    // Linear interpolation: y = vlo*(1-t) + vhi*t
    vlo := lut_table[lo];
    vhi := lut_table[hi];
    t := (x - lut_grid[lo]) / (lut_grid[hi] - lut_grid[lo] + 1.0E-10);
    "BsplineEval" := vlo * (1.0 - t) + vhi * t;
END_FUNCTION

FUNCTION_BLOCK "NeuroPLC_Inference"
{ S7_Optimized_Access := 'TRUE' }
VERSION : 0.1
VAR_INPUT
    features : Array[0..27] of Real;
END_VAR

VAR_OUTPUT
    fault_class : Int;
    confidence : Real;
END_VAR

VAR
    i, j, k : Int;
    sum_val, max_val, t_val : Real;
    v0 : Array[0..27] of Real;
    v1 : Array[0..27] of Real;
    v3 : Array[0..15, 0..27] of Real;
    v2 : Array[0..15] of Real;
    v4 : Array[0..15] of Real;
    v5 : Array[0..15] of Real;
    v7 : Array[0..3, 0..15] of Real;
    v6 : Array[0..3] of Real;
    v8 : Array[0..3] of Real;
    v9 : Array[0..3] of Real;
    lut_tmp : Array[0..14] of Real;
END_VAR

BEGIN
    // ---- Input ----
    FOR i := 0 TO 27 DO
        v0[i] := features[i];
    END_FOR;

    // ---- l0_silu: SILU ----
    v1[0] := v0[0] / (1.0 + EXP(-v0[0]));
    v1[1] := v0[1] / (1.0 + EXP(-v0[1]));
    v1[2] := v0[2] / (1.0 + EXP(-v0[2]));
    v1[3] := v0[3] / (1.0 + EXP(-v0[3]));
    v1[4] := v0[4] / (1.0 + EXP(-v0[4]));
    v1[5] := v0[5] / (1.0 + EXP(-v0[5]));
    v1[6] := v0[6] / (1.0 + EXP(-v0[6]));
    v1[7] := v0[7] / (1.0 + EXP(-v0[7]));
    v1[8] := v0[8] / (1.0 + EXP(-v0[8]));
    v1[9] := v0[9] / (1.0 + EXP(-v0[9]));
    v1[10] := v0[10] / (1.0 + EXP(-v0[10]));
    v1[11] := v0[11] / (1.0 + EXP(-v0[11]));
    v1[12] := v0[12] / (1.0 + EXP(-v0[12]));
    v1[13] := v0[13] / (1.0 + EXP(-v0[13]));
    v1[14] := v0[14] / (1.0 + EXP(-v0[14]));
    v1[15] := v0[15] / (1.0 + EXP(-v0[15]));
    v1[16] := v0[16] / (1.0 + EXP(-v0[16]));
    v1[17] := v0[17] / (1.0 + EXP(-v0[17]));
    v1[18] := v0[18] / (1.0 + EXP(-v0[18]));
    v1[19] := v0[19] / (1.0 + EXP(-v0[19]));
    v1[20] := v0[20] / (1.0 + EXP(-v0[20]));
    v1[21] := v0[21] / (1.0 + EXP(-v0[21]));
    v1[22] := v0[22] / (1.0 + EXP(-v0[22]));
    v1[23] := v0[23] / (1.0 + EXP(-v0[23]));
    v1[24] := v0[24] / (1.0 + EXP(-v0[24]));
    v1[25] := v0[25] / (1.0 + EXP(-v0[25]));
    v1[26] := v0[26] / (1.0 + EXP(-v0[26]));
    v1[27] := v0[27] / (1.0 + EXP(-v0[27]));

    // ---- l0_bspline: BsplineLUT(28×16, 15pts) ----
    // φ[0→0]: evaluate LUT (table offset 0)
    FOR k := 0 TO 14 DO
        lut_tmp[k] := "NeuroPLC_Weights".w1[0 + k];
    END_FOR;
    v3[0, 0] := "BsplineEval"(x := v0[0], lut_grid := "NeuroPLC_Weights".w0, lut_table := lut_tmp);
    // φ[1→0]: evaluate LUT (table offset 15)
    FOR k := 0 TO 14 DO
        lut_tmp[k] := "NeuroPLC_Weights".w1[15 + k];
    END_FOR;
    v3[0, 1] := "BsplineEval"(x := v0[1], lut_grid := "NeuroPLC_Weights".w0, lut_table := lut_tmp);
    // φ[2→0]: evaluate LUT (table offset 30)
    FOR k := 0 TO 14 DO
        lut_tmp[k] := "NeuroPLC_Weights".w1[30 + k];
    END_FOR;
    v3[0, 2] := "BsplineEval"(x := v0[2], lut_grid := "NeuroPLC_Weights".w0, lut_table := lut_tmp);
    // φ[3→0]: evaluate LUT (table offset 45)
    FOR k := 0 TO 14 DO
        lut_tmp[k] := "NeuroPLC_Weights".w1[45 + k];
    END_FOR;
    v3[0, 3] := "BsplineEval"(x := v0[3], lut_grid := "NeuroPLC_Weights".w0, lut_table := lut_tmp);
    // φ[4→0]: evaluate LUT (table offset 60)
    FOR k := 0 TO 14 DO
        lut_tmp[k] := "NeuroPLC_Weights".w1[60 + k];
    END_FOR;
    v3[0, 4] := "BsplineEval"(x := v0[4], lut_grid := "NeuroPLC_Weights".w0, lut_table := lut_tmp);
    // φ[5→0]: evaluate LUT (table offset 75)
    FOR k := 0 TO 14 DO
        lut_tmp[k] := "NeuroPLC_Weights".w1[75 + k];
    END_FOR;
    v3[0, 5] := "BsplineEval"(x := v0[5], lut_grid := "NeuroPLC_Weights".w0, lut_table := lut_tmp);
    // φ[6→0]: evaluate LUT (table offset 90)
    FOR k := 0 TO 14 DO
        lut_tmp[k] := "NeuroPLC_Weights".w1[90 + k];
    END_FOR;
    v3[0, 6] := "BsplineEval"(x := v0[6], lut_grid := "NeuroPLC_Weights".w0, lut_table := lut_tmp);
    // φ[7→0]: evaluate LUT (table offset 105)
    FOR k := 0 TO 14 DO
        lut_tmp[k] := "NeuroPLC_Weights".w1[105 + k];
    END_FOR;
    v3[0, 7] := "BsplineEval"(x := v0[7], lut_grid := "NeuroPLC_Weights".w0, lut_table := lut_tmp);
    // φ[8→0]: evaluate LUT (table offset 120)
    FOR k := 0 TO 14 DO
        lut_tmp[k] := "NeuroPLC_Weights".w1[120 + k];
    END_FOR;
    v3[0, 8] := "BsplineEval"(x := v0[8], lut_grid := "NeuroPLC_Weights".w0, lut_table := lut_tmp);
    // φ[9→0]: evaluate LUT (table offset 135)
    FOR k := 0 TO 14 DO
        lut_tmp[k] := "NeuroPLC_Weights".w1[135 + k];
    END_FOR;
    v3[0, 9] := "BsplineEval"(x := v0[9], lut_grid := "NeuroPLC_Weights".w0, lut_table := lut_tmp);
    // φ[10→0]: evaluate LUT (table offset 150)
    FOR k := 0 TO 14 DO
        lut_tmp[k] := "NeuroPLC_Weights".w1[150 + k];
    END_FOR;
    v3[0, 10] := "BsplineEval"(x := v0[10], lut_grid := "NeuroPLC_Weights".w0, lut_table := lut_tmp);
    // φ[11→0]: evaluate LUT (table offset 165)
    FOR k := 0 TO 14 DO
        lut_tmp[k] := "NeuroPLC_Weights".w1[165 + k];
    END_FOR;
    v3[0, 11] := "BsplineEval"(x := v0[11], lut_grid := "NeuroPLC_Weights".w0, lut_table := lut_tmp);
    // φ[12→0]: evaluate LUT (table offset 180)
    FOR k := 0 TO 14 DO
        lut_tmp[k] := "NeuroPLC_Weights".w1[180 + k];
    END_FOR;
    v3[0, 12] := "BsplineEval"(x := v0[12], lut_grid := "NeuroPLC_Weights".w0, lut_table := lut_tmp);
    // φ[13→0]: evaluate LUT (table offset 195)
    FOR k := 0 TO 14 DO
        lut_tmp[k] := "NeuroPLC_Weights".w1[195 + k];
    END_FOR;
    v3[0, 13] := "BsplineEval"(x := v0[13], lut_grid := "NeuroPLC_Weights".w0, lut_table := lut_tmp);
    // φ[14→0]: evaluate LUT (table offset 210)
    FOR k := 0 TO 14 DO
        lut_tmp[k] := "NeuroPLC_Weights".w1[210 + k];
    END_FOR;
    v3[0, 14] := "BsplineEval"(x := v0[14], lut_grid := "NeuroPLC_Weights".w0, lut_table := lut_tmp);
    // φ[15→0]: evaluate LUT (table offset 225)
    FOR k := 0 TO 14 DO
        lut_tmp[k] := "NeuroPLC_Weights".w1[225 + k];
    END_FOR;
    v3[0, 15] := "BsplineEval"(x := v0[15], lut_grid := "NeuroPLC_Weights".w0, lut_table := lut_tmp);
    // φ[16→0]: evaluate LUT (table offset 240)
    FOR k := 0 TO 14 DO
        lut_tmp[k] := "NeuroPLC_Weights".w1[240 + k];
    END_FOR;
    v3[0, 16] := "BsplineEval"(x := v0[16], lut_grid := "NeuroPLC_Weights".w0, lut_table := lut_tmp);
    // φ[17→0]: evaluate LUT (table offset 255)
    FOR k := 0 TO 14 DO
        lut_tmp[k] := "NeuroPLC_Weights".w1[255 + k];
    END_FOR;
    v3[0, 17] := "BsplineEval"(x := v0[17], lut_grid := "NeuroPLC_Weights".w0, lut_table := lut_tmp);
    // φ[18→0]: evaluate LUT (table offset 270)
    FOR k := 0 TO 14 DO
        lut_tmp[k] := "NeuroPLC_Weights".w1[270 + k];
    END_FOR;
    v3[0, 18] := "BsplineEval"(x := v0[18], lut_grid := "NeuroPLC_Weights".w0, lut_table := lut_tmp);
    // φ[19→0]: evaluate LUT (table offset 285)
    FOR k := 0 TO 14 DO
        lut_tmp[k] := "NeuroPLC_Weights".w1[285 + k];
    END_FOR;
    v3[0, 19] := "BsplineEval"(x := v0[19], lut_grid := "NeuroPLC_Weights".w0, lut_table := lut_tmp);
    // φ[20→0]: evaluate LUT (table offset 300)
    FOR k := 0 TO 14 DO
        lut_tmp[k] := "NeuroPLC_Weights".w1[300 + k];
    END_FOR;
    v3[0, 20] := "BsplineEval"(x := v0[20], lut_grid := "NeuroPLC_Weights".w0, lut_table := lut_tmp);
    // φ[21→0]: evaluate LUT (table offset 315)
    FOR k := 0 TO 14 DO
        lut_tmp[k] := "NeuroPLC_Weights".w1[315 + k];
    END_FOR;
    v3[0, 21] := "BsplineEval"(x := v0[21], lut_grid := "NeuroPLC_Weights".w0, lut_table := lut_tmp);
    // φ[22→0]: evaluate LUT (table offset 330)
    FOR k := 0 TO 14 DO
        lut_tmp[k] := "NeuroPLC_Weights".w1[330 + k];
    END_FOR;
    v3[0, 22] := "BsplineEval"(x := v0[22], lut_grid := "NeuroPLC_Weights".w0, lut_table := lut_tmp);
    // φ[23→0]: evaluate LUT (table offset 345)
    FOR k := 0 TO 14 DO
        lut_tmp[k] := "NeuroPLC_Weights".w1[345 + k];
    END_FOR;
    v3[0, 23] := "BsplineEval"(x := v0[23], lut_grid := "NeuroPLC_Weights".w0, lut_table := lut_tmp);
    // φ[24→0]: evaluate LUT (table offset 360)
    FOR k := 0 TO 14 DO
        lut_tmp[k] := "NeuroPLC_Weights".w1[360 + k];
    END_FOR;
    v3[0, 24] := "BsplineEval"(x := v0[24], lut_grid := "NeuroPLC_Weights".w0, lut_table := lut_tmp);
    // φ[25→0]: evaluate LUT (table offset 375)
    FOR k := 0 TO 14 DO
        lut_tmp[k] := "NeuroPLC_Weights".w1[375 + k];
    END_FOR;
    v3[0, 25] := "BsplineEval"(x := v0[25], lut_grid := "NeuroPLC_Weights".w0, lut_table := lut_tmp);
    // φ[26→0]: evaluate LUT (table offset 390)
    FOR k := 0 TO 14 DO
        lut_tmp[k] := "NeuroPLC_Weights".w1[390 + k];
    END_FOR;
    v3[0, 26] := "BsplineEval"(x := v0[26], lut_grid := "NeuroPLC_Weights".w0, lut_table := lut_tmp);
    // φ[27→0]: evaluate LUT (table offset 405)
    FOR k := 0 TO 14 DO
        lut_tmp[k] := "NeuroPLC_Weights".w1[405 + k];
    END_FOR;
    v3[0, 27] := "BsplineEval"(x := v0[27], lut_grid := "NeuroPLC_Weights".w0, lut_table := lut_tmp);
    // φ[0→1]: evaluate LUT (table offset 420)
    FOR k := 0 TO 14 DO
        lut_tmp[k] := "NeuroPLC_Weights".w1[420 + k];
    END_FOR;
    v3[1, 0] := "BsplineEval"(x := v0[0], lut_grid := "NeuroPLC_Weights".w0, lut_table := lut_tmp);
    // φ[1→1]: evaluate LUT (table offset 435)
    FOR k := 0 TO 14 DO
        lut_tmp[k] := "NeuroPLC_Weights".w1[435 + k];
    END_FOR;
    v3[1, 1] := "BsplineEval"(x := v0[1], lut_grid := "NeuroPLC_Weights".w0, lut_table := lut_tmp);
    // φ[2→1]: evaluate LUT (table offset 450)
    FOR k := 0 TO 14 DO
        lut_tmp[k] := "NeuroPLC_Weights".w1[450 + k];
    END_FOR;
    v3[1, 2] := "BsplineEval"(x := v0[2], lut_grid := "NeuroPLC_Weights".w0, lut_table := lut_tmp);
    // φ[3→1]: evaluate LUT (table offset 465)
    FOR k := 0 TO 14 DO
        lut_tmp[k] := "NeuroPLC_Weights".w1[465 + k];
    END_FOR;
    v3[1, 3] := "BsplineEval"(x := v0[3], lut_grid := "NeuroPLC_Weights".w0, lut_table := lut_tmp);
    // φ[4→1]: evaluate LUT (table offset 480)
    FOR k := 0 TO 14 DO
        lut_tmp[k] := "NeuroPLC_Weights".w1[480 + k];
    END_FOR;
    v3[1, 4] := "BsplineEval"(x := v0[4], lut_grid := "NeuroPLC_Weights".w0, lut_table := lut_tmp);
    // φ[5→1]: evaluate LUT (table offset 495)
    FOR k := 0 TO 14 DO
        lut_tmp[k] := "NeuroPLC_Weights".w1[495 + k];
    END_FOR;
    v3[1, 5] := "BsplineEval"(x := v0[5], lut_grid := "NeuroPLC_Weights".w0, lut_table := lut_tmp);
    // φ[6→1]: evaluate LUT (table offset 510)
    FOR k := 0 TO 14 DO
        lut_tmp[k] := "NeuroPLC_Weights".w1[510 + k];
    END_FOR;
    v3[1, 6] := "BsplineEval"(x := v0[6], lut_grid := "NeuroPLC_Weights".w0, lut_table := lut_tmp);
    // φ[7→1]: evaluate LUT (table offset 525)
    FOR k := 0 TO 14 DO
        lut_tmp[k] := "NeuroPLC_Weights".w1[525 + k];
    END_FOR;
    v3[1, 7] := "BsplineEval"(x := v0[7], lut_grid := "NeuroPLC_Weights".w0, lut_table := lut_tmp);
    // φ[8→1]: evaluate LUT (table offset 540)
    FOR k := 0 TO 14 DO
        lut_tmp[k] := "NeuroPLC_Weights".w1[540 + k];
    END_FOR;
    v3[1, 8] := "BsplineEval"(x := v0[8], lut_grid := "NeuroPLC_Weights".w0, lut_table := lut_tmp);
    // φ[9→1]: evaluate LUT (table offset 555)
    FOR k := 0 TO 14 DO
        lut_tmp[k] := "NeuroPLC_Weights".w1[555 + k];
    END_FOR;
    v3[1, 9] := "BsplineEval"(x := v0[9], lut_grid := "NeuroPLC_Weights".w0, lut_table := lut_tmp);
    // φ[10→1]: evaluate LUT (table offset 570)
    FOR k := 0 TO 14 DO
        lut_tmp[k] := "NeuroPLC_Weights".w1[570 + k];
    END_FOR;
    v3[1, 10] := "BsplineEval"(x := v0[10], lut_grid := "NeuroPLC_Weights".w0, lut_table := lut_tmp);
    // φ[11→1]: evaluate LUT (table offset 585)
    FOR k := 0 TO 14 DO
        lut_tmp[k] := "NeuroPLC_Weights".w1[585 + k];
    END_FOR;
    v3[1, 11] := "BsplineEval"(x := v0[11], lut_grid := "NeuroPLC_Weights".w0, lut_table := lut_tmp);
    // φ[12→1]: evaluate LUT (table offset 600)
    FOR k := 0 TO 14 DO
        lut_tmp[k] := "NeuroPLC_Weights".w1[600 + k];
    END_FOR;
    v3[1, 12] := "BsplineEval"(x := v0[12], lut_grid := "NeuroPLC_Weights".w0, lut_table := lut_tmp);
    // φ[13→1]: evaluate LUT (table offset 615)
    FOR k := 0 TO 14 DO
        lut_tmp[k] := "NeuroPLC_Weights".w1[615 + k];
    END_FOR;
    v3[1, 13] := "BsplineEval"(x := v0[13], lut_grid := "NeuroPLC_Weights".w0, lut_table := lut_tmp);
    // φ[14→1]: evaluate LUT (table offset 630)
    FOR k := 0 TO 14 DO
        lut_tmp[k] := "NeuroPLC_Weights".w1[630 + k];
    END_FOR;
    v3[1, 14] := "BsplineEval"(x := v0[14], lut_grid := "NeuroPLC_Weights".w0, lut_table := lut_tmp);
    // φ[15→1]: evaluate LUT (table offset 645)
    FOR k := 0 TO 14 DO
        lut_tmp[k] := "NeuroPLC_Weights".w1[645 + k];
    END_FOR;
    v3[1, 15] := "BsplineEval"(x := v0[15], lut_grid := "NeuroPLC_Weights".w0, lut_table := lut_tmp);
    // φ[16→1]: evaluate LUT (table offset 660)
    FOR k := 0 TO 14 DO
        lut_tmp[k] := "NeuroPLC_Weights".w1[660 + k];
    END_FOR;
    v3[1, 16] := "BsplineEval"(x := v0[16], lut_grid := "NeuroPLC_Weights".w0, lut_table := lut_tmp);
    // φ[17→1]: evaluate LUT (table offset 675)
    FOR k := 0 TO 14 DO
        lut_tmp[k] := "NeuroPLC_Weights".w1[675 + k];
    END_FOR;
    v3[1, 17] := "BsplineEval"(x := v0[17], lut_grid := "NeuroPLC_Weights".w0, lut_table := lut_tmp);
    // φ[18→1]: evaluate LUT (table offset 690)
    FOR k := 0 TO 14 DO
        lut_tmp[k] := "NeuroPLC_Weights".w1[690 + k];
    END_FOR;
    v3[1, 18] := "BsplineEval"(x := v0[18], lut_grid := "NeuroPLC_Weights".w0, lut_table := lut_tmp);
    // φ[19→1]: evaluate LUT (table offset 705)
    FOR k := 0 TO 14 DO
        lut_tmp[k] := "NeuroPLC_Weights".w1[705 + k];
    END_FOR;
    v3[1, 19] := "BsplineEval"(x := v0[19], lut_grid := "NeuroPLC_Weights".w0, lut_table := lut_tmp);
    // φ[20→1]: evaluate LUT (table offset 720)
    FOR k := 0 TO 14 DO
        lut_tmp[k] := "NeuroPLC_Weights".w1[720 + k];
    END_FOR;
    v3[1, 20] := "BsplineEval"(x := v0[20], lut_grid := "NeuroPLC_Weights".w0, lut_table := lut_tmp);
    // φ[21→1]: evaluate LUT (table offset 735)
    FOR k := 0 TO 14 DO
        lut_tmp[k] := "NeuroPLC_Weights".w1[735 + k];
    END_FOR;
    v3[1, 21] := "BsplineEval"(x := v0[21], lut_grid := "NeuroPLC_Weights".w0, lut_table := lut_tmp);
    // φ[22→1]: evaluate LUT (table offset 750)
    FOR k := 0 TO 14 DO
        lut_tmp[k] := "NeuroPLC_Weights".w1[750 + k];
    END_FOR;
    v3[1, 22] := "BsplineEval"(x := v0[22], lut_grid := "NeuroPLC_Weights".w0, lut_table := lut_tmp);
    // φ[23→1]: evaluate LUT (table offset 765)
    FOR k := 0 TO 14 DO
        lut_tmp[k] := "NeuroPLC_Weights".w1[765 + k];
    END_FOR;
    v3[1, 23] := "BsplineEval"(x := v0[23], lut_grid := "NeuroPLC_Weights".w0, lut_table := lut_tmp);
    // φ[24→1]: evaluate LUT (table offset 780)
    FOR k := 0 TO 14 DO
        lut_tmp[k] := "NeuroPLC_Weights".w1[780 + k];
    END_FOR;
    v3[1, 24] := "BsplineEval"(x := v0[24], lut_grid := "NeuroPLC_Weights".w0, lut_table := lut_tmp);
    // φ[25→1]: evaluate LUT (table offset 795)
    FOR k := 0 TO 14 DO
        lut_tmp[k] := "NeuroPLC_Weights".w1[795 + k];
    END_FOR;
    v3[1, 25] := "BsplineEval"(x := v0[25], lut_grid := "NeuroPLC_Weights".w0, lut_table := lut_tmp);
    // φ[26→1]: evaluate LUT (table offset 810)
    FOR k := 0 TO 14 DO
        lut_tmp[k] := "NeuroPLC_Weights".w1[810 + k];
    END_FOR;
    v3[1, 26] := "BsplineEval"(x := v0[26], lut_grid := "NeuroPLC_Weights".w0, lut_table := lut_tmp);
    // φ[27→1]: evaluate LUT (table offset 825)
    FOR k := 0 TO 14 DO
        lut_tmp[k] := "NeuroPLC_Weights".w1[825 + k];
    END_FOR;
    v3[1, 27] := "BsplineEval"(x := v0[27], lut_grid := "NeuroPLC_Weights".w0, lut_table := lut_tmp);
    // φ[0→2]: evaluate LUT (table offset 840)
    FOR k := 0 TO 14 DO
        lut_tmp[k] := "NeuroPLC_Weights".w1[840 + k];
    END_FOR;
    v3[2, 0] := "BsplineEval"(x := v0[0], lut_grid := "NeuroPLC_Weights".w0, lut_table := lut_tmp);
    // φ[1→2]: evaluate LUT (table offset 855)
    FOR k := 0 TO 14 DO
        lut_tmp[k] := "NeuroPLC_Weights".w1[855 + k];
    END_FOR;
    v3[2, 1] := "BsplineEval"(x := v0[1], lut_grid := "NeuroPLC_Weights".w0, lut_table := lut_tmp);
    // φ[2→2]: evaluate LUT (table offset 870)
    FOR k := 0 TO 14 DO
        lut_tmp[k] := "NeuroPLC_Weights".w1[870 + k];
    END_FOR;
    v3[2, 2] := "BsplineEval"(x := v0[2], lut_grid := "NeuroPLC_Weights".w0, lut_table := lut_tmp);
    // φ[3→2]: evaluate LUT (table offset 885)
    FOR k := 0 TO 14 DO
        lut_tmp[k] := "NeuroPLC_Weights".w1[885 + k];
    END_FOR;
    v3[2, 3] := "BsplineEval"(x := v0[3], lut_grid := "NeuroPLC_Weights".w0, lut_table := lut_tmp);
    // φ[4→2]: evaluate LUT (table offset 900)
    FOR k := 0 TO 14 DO
        lut_tmp[k] := "NeuroPLC_Weights".w1[900 + k];
    END_FOR;
    v3[2, 4] := "BsplineEval"(x := v0[4], lut_grid := "NeuroPLC_Weights".w0, lut_table := lut_tmp);
    // φ[5→2]: evaluate LUT (table offset 915)
    FOR k := 0 TO 14 DO
        lut_tmp[k] := "NeuroPLC_Weights".w1[915 + k];
    END_FOR;
    v3[2, 5] := "BsplineEval"(x := v0[5], lut_grid := "NeuroPLC_Weights".w0, lut_table := lut_tmp);
    // φ[6→2]: evaluate LUT (table offset 930)
    FOR k := 0 TO 14 DO
        lut_tmp[k] := "NeuroPLC_Weights".w1[930 + k];
    END_FOR;
    v3[2, 6] := "BsplineEval"(x := v0[6], lut_grid := "NeuroPLC_Weights".w0, lut_table := lut_tmp);
    // φ[7→2]: evaluate LUT (table offset 945)
    FOR k := 0 TO 14 DO
        lut_tmp[k] := "NeuroPLC_Weights".w1[945 + k];
    END_FOR;
    v3[2, 7] := "BsplineEval"(x := v0[7], lut_grid := "NeuroPLC_Weights".w0, lut_table := lut_tmp);
    // φ[8→2]: evaluate LUT (table offset 960)
    FOR k := 0 TO 14 DO
        lut_tmp[k] := "NeuroPLC_Weights".w1[960 + k];
    END_FOR;
    v3[2, 8] := "BsplineEval"(x := v0[8], lut_grid := "NeuroPLC_Weights".w0, lut_table := lut_tmp);
    // φ[9→2]: evaluate LUT (table offset 975)
    FOR k := 0 TO 14 DO
        lut_tmp[k] := "NeuroPLC_Weights".w1[975 + k];
    END_FOR;
    v3[2, 9] := "BsplineEval"(x := v0[9], lut_grid := "NeuroPLC_Weights".w0, lut_table := lut_tmp);
    // φ[10→2]: evaluate LUT (table offset 990)
    FOR k := 0 TO 14 DO
        lut_tmp[k] := "NeuroPLC_Weights".w1[990 + k];
    END_FOR;
    v3[2, 10] := "BsplineEval"(x := v0[10], lut_grid := "NeuroPLC_Weights".w0, lut_table := lut_tmp);
    // φ[11→2]: evaluate LUT (table offset 1005)
    FOR k := 0 TO 14 DO
        lut_tmp[k] := "NeuroPLC_Weights".w1[1005 + k];
    END_FOR;
    v3[2, 11] := "BsplineEval"(x := v0[11], lut_grid := "NeuroPLC_Weights".w0, lut_table := lut_tmp);
    // φ[12→2]: evaluate LUT (table offset 1020)
    FOR k := 0 TO 14 DO
        lut_tmp[k] := "NeuroPLC_Weights".w1[1020 + k];
    END_FOR;
    v3[2, 12] := "BsplineEval"(x := v0[12], lut_grid := "NeuroPLC_Weights".w0, lut_table := lut_tmp);
    // φ[13→2]: evaluate LUT (table offset 1035)
    FOR k := 0 TO 14 DO
        lut_tmp[k] := "NeuroPLC_Weights".w1[1035 + k];
    END_FOR;
    v3[2, 13] := "BsplineEval"(x := v0[13], lut_grid := "NeuroPLC_Weights".w0, lut_table := lut_tmp);
    // φ[14→2]: evaluate LUT (table offset 1050)
    FOR k := 0 TO 14 DO
        lut_tmp[k] := "NeuroPLC_Weights".w1[1050 + k];
    END_FOR;
    v3[2, 14] := "BsplineEval"(x := v0[14], lut_grid := "NeuroPLC_Weights".w0, lut_table := lut_tmp);
    // φ[15→2]: evaluate LUT (table offset 1065)
    FOR k := 0 TO 14 DO
        lut_tmp[k] := "NeuroPLC_Weights".w1[1065 + k];
    END_FOR;
    v3[2, 15] := "BsplineEval"(x := v0[15], lut_grid := "NeuroPLC_Weights".w0, lut_table := lut_tmp);
    // φ[16→2]: evaluate LUT (table offset 1080)
    FOR k := 0 TO 14 DO
        lut_tmp[k] := "NeuroPLC_Weights".w1[1080 + k];
    END_FOR;
    v3[2, 16] := "BsplineEval"(x := v0[16], lut_grid := "NeuroPLC_Weights".w0, lut_table := lut_tmp);
    // φ[17→2]: evaluate LUT (table offset 1095)
    FOR k := 0 TO 14 DO
        lut_tmp[k] := "NeuroPLC_Weights".w1[1095 + k];
    END_FOR;
    v3[2, 17] := "BsplineEval"(x := v0[17], lut_grid := "NeuroPLC_Weights".w0, lut_table := lut_tmp);
    // φ[18→2]: evaluate LUT (table offset 1110)
    FOR k := 0 TO 14 DO
        lut_tmp[k] := "NeuroPLC_Weights".w1[1110 + k];
    END_FOR;
    v3[2, 18] := "BsplineEval"(x := v0[18], lut_grid := "NeuroPLC_Weights".w0, lut_table := lut_tmp);
    // φ[19→2]: evaluate LUT (table offset 1125)
    FOR k := 0 TO 14 DO
        lut_tmp[k] := "NeuroPLC_Weights".w1[1125 + k];
    END_FOR;
    v3[2, 19] := "BsplineEval"(x := v0[19], lut_grid := "NeuroPLC_Weights".w0, lut_table := lut_tmp);
    // φ[20→2]: evaluate LUT (table offset 1140)
    FOR k := 0 TO 14 DO
        lut_tmp[k] := "NeuroPLC_Weights".w1[1140 + k];
    END_FOR;
    v3[2, 20] := "BsplineEval"(x := v0[20], lut_grid := "NeuroPLC_Weights".w0, lut_table := lut_tmp);
    // φ[21→2]: evaluate LUT (table offset 1155)
    FOR k := 0 TO 14 DO
        lut_tmp[k] := "NeuroPLC_Weights".w1[1155 + k];
    END_FOR;
    v3[2, 21] := "BsplineEval"(x := v0[21], lut_grid := "NeuroPLC_Weights".w0, lut_table := lut_tmp);
    // φ[22→2]: evaluate LUT (table offset 1170)
    FOR k := 0 TO 14 DO
        lut_tmp[k] := "NeuroPLC_Weights".w1[1170 + k];
    END_FOR;
    v3[2, 22] := "BsplineEval"(x := v0[22], lut_grid := "NeuroPLC_Weights".w0, lut_table := lut_tmp);
    // φ[23→2]: evaluate LUT (table offset 1185)
    FOR k := 0 TO 14 DO
        lut_tmp[k] := "NeuroPLC_Weights".w1[1185 + k];
    END_FOR;
    v3[2, 23] := "BsplineEval"(x := v0[23], lut_grid := "NeuroPLC_Weights".w0, lut_table := lut_tmp);
    // φ[24→2]: evaluate LUT (table offset 1200)
    FOR k := 0 TO 14 DO
        lut_tmp[k] := "NeuroPLC_Weights".w1[1200 + k];
    END_FOR;
    v3[2, 24] := "BsplineEval"(x := v0[24], lut_grid := "NeuroPLC_Weights".w0, lut_table := lut_tmp);
    // φ[25→2]: evaluate LUT (table offset 1215)
    FOR k := 0 TO 14 DO
        lut_tmp[k] := "NeuroPLC_Weights".w1[1215 + k];
    END_FOR;
    v3[2, 25] := "BsplineEval"(x := v0[25], lut_grid := "NeuroPLC_Weights".w0, lut_table := lut_tmp);
    // φ[26→2]: evaluate LUT (table offset 1230)
    FOR k := 0 TO 14 DO
        lut_tmp[k] := "NeuroPLC_Weights".w1[1230 + k];
    END_FOR;
    v3[2, 26] := "BsplineEval"(x := v0[26], lut_grid := "NeuroPLC_Weights".w0, lut_table := lut_tmp);
    // φ[27→2]: evaluate LUT (table offset 1245)
    FOR k := 0 TO 14 DO
        lut_tmp[k] := "NeuroPLC_Weights".w1[1245 + k];
    END_FOR;
    v3[2, 27] := "BsplineEval"(x := v0[27], lut_grid := "NeuroPLC_Weights".w0, lut_table := lut_tmp);
    // φ[0→3]: evaluate LUT (table offset 1260)
    FOR k := 0 TO 14 DO
        lut_tmp[k] := "NeuroPLC_Weights".w1[1260 + k];
    END_FOR;
    v3[3, 0] := "BsplineEval"(x := v0[0], lut_grid := "NeuroPLC_Weights".w0, lut_table := lut_tmp);
    // φ[1→3]: evaluate LUT (table offset 1275)
    FOR k := 0 TO 14 DO
        lut_tmp[k] := "NeuroPLC_Weights".w1[1275 + k];
    END_FOR;
    v3[3, 1] := "BsplineEval"(x := v0[1], lut_grid := "NeuroPLC_Weights".w0, lut_table := lut_tmp);
    // φ[2→3]: evaluate LUT (table offset 1290)
    FOR k := 0 TO 14 DO
        lut_tmp[k] := "NeuroPLC_Weights".w1[1290 + k];
    END_FOR;
    v3[3, 2] := "BsplineEval"(x := v0[2], lut_grid := "NeuroPLC_Weights".w0, lut_table := lut_tmp);
    // φ[3→3]: evaluate LUT (table offset 1305)
    FOR k := 0 TO 14 DO
        lut_tmp[k] := "NeuroPLC_Weights".w1[1305 + k];
    END_FOR;
    v3[3, 3] := "BsplineEval"(x := v0[3], lut_grid := "NeuroPLC_Weights".w0, lut_table := lut_tmp);
    // φ[4→3]: evaluate LUT (table offset 1320)
    FOR k := 0 TO 14 DO
        lut_tmp[k] := "NeuroPLC_Weights".w1[1320 + k];
    END_FOR;
    v3[3, 4] := "BsplineEval"(x := v0[4], lut_grid := "NeuroPLC_Weights".w0, lut_table := lut_tmp);
    // φ[5→3]: evaluate LUT (table offset 1335)
    FOR k := 0 TO 14 DO
        lut_tmp[k] := "NeuroPLC_Weights".w1[1335 + k];
    END_FOR;
    v3[3, 5] := "BsplineEval"(x := v0[5], lut_grid := "NeuroPLC_Weights".w0, lut_table := lut_tmp);
    // φ[6→3]: evaluate LUT (table offset 1350)
    FOR k := 0 TO 14 DO
        lut_tmp[k] := "NeuroPLC_Weights".w1[1350 + k];
    END_FOR;
    v3[3, 6] := "BsplineEval"(x := v0[6], lut_grid := "NeuroPLC_Weights".w0, lut_table := lut_tmp);
    // φ[7→3]: evaluate LUT (table offset 1365)
    FOR k := 0 TO 14 DO
        lut_tmp[k] := "NeuroPLC_Weights".w1[1365 + k];
    END_FOR;
    v3[3, 7] := "BsplineEval"(x := v0[7], lut_grid := "NeuroPLC_Weights".w0, lut_table := lut_tmp);
    // φ[8→3]: evaluate LUT (table offset 1380)
    FOR k := 0 TO 14 DO
        lut_tmp[k] := "NeuroPLC_Weights".w1[1380 + k];
    END_FOR;
    v3[3, 8] := "BsplineEval"(x := v0[8], lut_grid := "NeuroPLC_Weights".w0, lut_table := lut_tmp);
    // φ[9→3]: evaluate LUT (table offset 1395)
    FOR k := 0 TO 14 DO
        lut_tmp[k] := "NeuroPLC_Weights".w1[1395 + k];
    END_FOR;
    v3[3, 9] := "BsplineEval"(x := v0[9], lut_grid := "NeuroPLC_Weights".w0, lut_table := lut_tmp);
    // φ[10→3]: evaluate LUT (table offset 1410)
    FOR k := 0 TO 14 DO
        lut_tmp[k] := "NeuroPLC_Weights".w1[1410 + k];
    END_FOR;
    v3[3, 10] := "BsplineEval"(x := v0[10], lut_grid := "NeuroPLC_Weights".w0, lut_table := lut_tmp);
    // φ[11→3]: evaluate LUT (table offset 1425)
    FOR k := 0 TO 14 DO
        lut_tmp[k] := "NeuroPLC_Weights".w1[1425 + k];
    END_FOR;
    v3[3, 11] := "BsplineEval"(x := v0[11], lut_grid := "NeuroPLC_Weights".w0, lut_table := lut_tmp);
    // φ[12→3]: evaluate LUT (table offset 1440)
    FOR k := 0 TO 14 DO
        lut_tmp[k] := "NeuroPLC_Weights".w1[1440 + k];
    END_FOR;
    v3[3, 12] := "BsplineEval"(x := v0[12], lut_grid := "NeuroPLC_Weights".w0, lut_table := lut_tmp);
    // φ[13→3]: evaluate LUT (table offset 1455)
    FOR k := 0 TO 14 DO
        lut_tmp[k] := "NeuroPLC_Weights".w1[1455 + k];
    END_FOR;
    v3[3, 13] := "BsplineEval"(x := v0[13], lut_grid := "NeuroPLC_Weights".w0, lut_table := lut_tmp);
    // φ[14→3]: evaluate LUT (table offset 1470)
    FOR k := 0 TO 14 DO
        lut_tmp[k] := "NeuroPLC_Weights".w1[1470 + k];
    END_FOR;
    v3[3, 14] := "BsplineEval"(x := v0[14], lut_grid := "NeuroPLC_Weights".w0, lut_table := lut_tmp);
    // φ[15→3]: evaluate LUT (table offset 1485)
    FOR k := 0 TO 14 DO
        lut_tmp[k] := "NeuroPLC_Weights".w1[1485 + k];
    END_FOR;
    v3[3, 15] := "BsplineEval"(x := v0[15], lut_grid := "NeuroPLC_Weights".w0, lut_table := lut_tmp);
    // φ[16→3]: evaluate LUT (table offset 1500)
    FOR k := 0 TO 14 DO
        lut_tmp[k] := "NeuroPLC_Weights".w1[1500 + k];
    END_FOR;
    v3[3, 16] := "BsplineEval"(x := v0[16], lut_grid := "NeuroPLC_Weights".w0, lut_table := lut_tmp);
    // φ[17→3]: evaluate LUT (table offset 1515)
    FOR k := 0 TO 14 DO
        lut_tmp[k] := "NeuroPLC_Weights".w1[1515 + k];
    END_FOR;
    v3[3, 17] := "BsplineEval"(x := v0[17], lut_grid := "NeuroPLC_Weights".w0, lut_table := lut_tmp);
    // φ[18→3]: evaluate LUT (table offset 1530)
    FOR k := 0 TO 14 DO
        lut_tmp[k] := "NeuroPLC_Weights".w1[1530 + k];
    END_FOR;
    v3[3, 18] := "BsplineEval"(x := v0[18], lut_grid := "NeuroPLC_Weights".w0, lut_table := lut_tmp);
    // φ[19→3]: evaluate LUT (table offset 1545)
    FOR k := 0 TO 14 DO
        lut_tmp[k] := "NeuroPLC_Weights".w1[1545 + k];
    END_FOR;
    v3[3, 19] := "BsplineEval"(x := v0[19], lut_grid := "NeuroPLC_Weights".w0, lut_table := lut_tmp);
    // φ[20→3]: evaluate LUT (table offset 1560)
    FOR k := 0 TO 14 DO
        lut_tmp[k] := "NeuroPLC_Weights".w1[1560 + k];
    END_FOR;
    v3[3, 20] := "BsplineEval"(x := v0[20], lut_grid := "NeuroPLC_Weights".w0, lut_table := lut_tmp);
    // φ[21→3]: evaluate LUT (table offset 1575)
    FOR k := 0 TO 14 DO
        lut_tmp[k] := "NeuroPLC_Weights".w1[1575 + k];
    END_FOR;
    v3[3, 21] := "BsplineEval"(x := v0[21], lut_grid := "NeuroPLC_Weights".w0, lut_table := lut_tmp);
    // φ[22→3]: evaluate LUT (table offset 1590)
    FOR k := 0 TO 14 DO
        lut_tmp[k] := "NeuroPLC_Weights".w1[1590 + k];
    END_FOR;
    v3[3, 22] := "BsplineEval"(x := v0[22], lut_grid := "NeuroPLC_Weights".w0, lut_table := lut_tmp);
    // φ[23→3]: evaluate LUT (table offset 1605)
    FOR k := 0 TO 14 DO
        lut_tmp[k] := "NeuroPLC_Weights".w1[1605 + k];
    END_FOR;
    v3[3, 23] := "BsplineEval"(x := v0[23], lut_grid := "NeuroPLC_Weights".w0, lut_table := lut_tmp);
    // φ[24→3]: evaluate LUT (table offset 1620)
    FOR k := 0 TO 14 DO
        lut_tmp[k] := "NeuroPLC_Weights".w1[1620 + k];
    END_FOR;
    v3[3, 24] := "BsplineEval"(x := v0[24], lut_grid := "NeuroPLC_Weights".w0, lut_table := lut_tmp);
    // φ[25→3]: evaluate LUT (table offset 1635)
    FOR k := 0 TO 14 DO
        lut_tmp[k] := "NeuroPLC_Weights".w1[1635 + k];
    END_FOR;
    v3[3, 25] := "BsplineEval"(x := v0[25], lut_grid := "NeuroPLC_Weights".w0, lut_table := lut_tmp);
    // φ[26→3]: evaluate LUT (table offset 1650)
    FOR k := 0 TO 14 DO
        lut_tmp[k] := "NeuroPLC_Weights".w1[1650 + k];
    END_FOR;
    v3[3, 26] := "BsplineEval"(x := v0[26], lut_grid := "NeuroPLC_Weights".w0, lut_table := lut_tmp);
    // φ[27→3]: evaluate LUT (table offset 1665)
    FOR k := 0 TO 14 DO
        lut_tmp[k] := "NeuroPLC_Weights".w1[1665 + k];
    END_FOR;
    v3[3, 27] := "BsplineEval"(x := v0[27], lut_grid := "NeuroPLC_Weights".w0, lut_table := lut_tmp);
    // φ[0→4]: evaluate LUT (table offset 1680)
    FOR k := 0 TO 14 DO
        lut_tmp[k] := "NeuroPLC_Weights".w1[1680 + k];
    END_FOR;
    v3[4, 0] := "BsplineEval"(x := v0[0], lut_grid := "NeuroPLC_Weights".w0, lut_table := lut_tmp);
    // φ[1→4]: evaluate LUT (table offset 1695)
    FOR k := 0 TO 14 DO
        lut_tmp[k] := "NeuroPLC_Weights".w1[1695 + k];
    END_FOR;
    v3[4, 1] := "BsplineEval"(x := v0[1], lut_grid := "NeuroPLC_Weights".w0, lut_table := lut_tmp);
    // φ[2→4]: evaluate LUT (table offset 1710)
    FOR k := 0 TO 14 DO
        lut_tmp[k] := "NeuroPLC_Weights".w1[1710 + k];
    END_FOR;
    v3[4, 2] := "BsplineEval"(x := v0[2], lut_grid := "NeuroPLC_Weights".w0, lut_table := lut_tmp);
    // φ[3→4]: evaluate LUT (table offset 1725)
    FOR k := 0 TO 14 DO
        lut_tmp[k] := "NeuroPLC_Weights".w1[1725 + k];
    END_FOR;
    v3[4, 3] := "BsplineEval"(x := v0[3], lut_grid := "NeuroPLC_Weights".w0, lut_table := lut_tmp);
    // φ[4→4]: evaluate LUT (table offset 1740)
    FOR k := 0 TO 14 DO
        lut_tmp[k] := "NeuroPLC_Weights".w1[1740 + k];
    END_FOR;
    v3[4, 4] := "BsplineEval"(x := v0[4], lut_grid := "NeuroPLC_Weights".w0, lut_table := lut_tmp);
    // φ[5→4]: evaluate LUT (table offset 1755)
    FOR k := 0 TO 14 DO
        lut_tmp[k] := "NeuroPLC_Weights".w1[1755 + k];
    END_FOR;
    v3[4, 5] := "BsplineEval"(x := v0[5], lut_grid := "NeuroPLC_Weights".w0, lut_table := lut_tmp);
    // φ[6→4]: evaluate LUT (table offset 1770)
    FOR k := 0 TO 14 DO
        lut_tmp[k] := "NeuroPLC_Weights".w1[1770 + k];
    END_FOR;
    v3[4, 6] := "BsplineEval"(x := v0[6], lut_grid := "NeuroPLC_Weights".w0, lut_table := lut_tmp);
    // φ[7→4]: evaluate LUT (table offset 1785)
    FOR k := 0 TO 14 DO
        lut_tmp[k] := "NeuroPLC_Weights".w1[1785 + k];
    END_FOR;
    v3[4, 7] := "BsplineEval"(x := v0[7], lut_grid := "NeuroPLC_Weights".w0, lut_table := lut_tmp);
    // φ[8→4]: evaluate LUT (table offset 1800)
    FOR k := 0 TO 14 DO
        lut_tmp[k] := "NeuroPLC_Weights".w1[1800 + k];
    END_FOR;
    v3[4, 8] := "BsplineEval"(x := v0[8], lut_grid := "NeuroPLC_Weights".w0, lut_table := lut_tmp);
    // φ[9→4]: evaluate LUT (table offset 1815)
    FOR k := 0 TO 14 DO
        lut_tmp[k] := "NeuroPLC_Weights".w1[1815 + k];
    END_FOR;
    v3[4, 9] := "BsplineEval"(x := v0[9], lut_grid := "NeuroPLC_Weights".w0, lut_table := lut_tmp);
    // φ[10→4]: evaluate LUT (table offset 1830)
    FOR k := 0 TO 14 DO
        lut_tmp[k] := "NeuroPLC_Weights".w1[1830 + k];
    END_FOR;
    v3[4, 10] := "BsplineEval"(x := v0[10], lut_grid := "NeuroPLC_Weights".w0, lut_table := lut_tmp);
    // φ[11→4]: evaluate LUT (table offset 1845)
    FOR k := 0 TO 14 DO
        lut_tmp[k] := "NeuroPLC_Weights".w1[1845 + k];
    END_FOR;
    v3[4, 11] := "BsplineEval"(x := v0[11], lut_grid := "NeuroPLC_Weights".w0, lut_table := lut_tmp);
    // φ[12→4]: evaluate LUT (table offset 1860)
    FOR k := 0 TO 14 DO
        lut_tmp[k] := "NeuroPLC_Weights".w1[1860 + k];
    END_FOR;
    v3[4, 12] := "BsplineEval"(x := v0[12], lut_grid := "NeuroPLC_Weights".w0, lut_table := lut_tmp);
    // φ[13→4]: evaluate LUT (table offset 1875)
    FOR k := 0 TO 14 DO
        lut_tmp[k] := "NeuroPLC_Weights".w1[1875 + k];
    END_FOR;
    v3[4, 13] := "BsplineEval"(x := v0[13], lut_grid := "NeuroPLC_Weights".w0, lut_table := lut_tmp);
    // φ[14→4]: evaluate LUT (table offset 1890)
    FOR k := 0 TO 14 DO
        lut_tmp[k] := "NeuroPLC_Weights".w1[1890 + k];
    END_FOR;
    v3[4, 14] := "BsplineEval"(x := v0[14], lut_grid := "NeuroPLC_Weights".w0, lut_table := lut_tmp);
    // φ[15→4]: evaluate LUT (table offset 1905)
    FOR k := 0 TO 14 DO
        lut_tmp[k] := "NeuroPLC_Weights".w1[1905 + k];
    END_FOR;
    v3[4, 15] := "BsplineEval"(x := v0[15], lut_grid := "NeuroPLC_Weights".w0, lut_table := lut_tmp);
    // φ[16→4]: evaluate LUT (table offset 1920)
    FOR k := 0 TO 14 DO
        lut_tmp[k] := "NeuroPLC_Weights".w1[1920 + k];
    END_FOR;
    v3[4, 16] := "BsplineEval"(x := v0[16], lut_grid := "NeuroPLC_Weights".w0, lut_table := lut_tmp);
    // φ[17→4]: evaluate LUT (table offset 1935)
    FOR k := 0 TO 14 DO
        lut_tmp[k] := "NeuroPLC_Weights".w1[1935 + k];
    END_FOR;
    v3[4, 17] := "BsplineEval"(x := v0[17], lut_grid := "NeuroPLC_Weights".w0, lut_table := lut_tmp);
    // φ[18→4]: evaluate LUT (table offset 1950)
    FOR k := 0 TO 14 DO
        lut_tmp[k] := "NeuroPLC_Weights".w1[1950 + k];
    END_FOR;
    v3[4, 18] := "BsplineEval"(x := v0[18], lut_grid := "NeuroPLC_Weights".w0, lut_table := lut_tmp);
    // φ[19→4]: evaluate LUT (table offset 1965)
    FOR k := 0 TO 14 DO
        lut_tmp[k] := "NeuroPLC_Weights".w1[1965 + k];
    END_FOR;
    v3[4, 19] := "BsplineEval"(x := v0[19], lut_grid := "NeuroPLC_Weights".w0, lut_table := lut_tmp);
    // φ[20→4]: evaluate LUT (table offset 1980)
    FOR k := 0 TO 14 DO
        lut_tmp[k] := "NeuroPLC_Weights".w1[1980 + k];
    END_FOR;
    v3[4, 20] := "BsplineEval"(x := v0[20], lut_grid := "NeuroPLC_Weights".w0, lut_table := lut_tmp);
    // φ[21→4]: evaluate LUT (table offset 1995)
    FOR k := 0 TO 14 DO
        lut_tmp[k] := "NeuroPLC_Weights".w1[1995 + k];
    END_FOR;
    v3[4, 21] := "BsplineEval"(x := v0[21], lut_grid := "NeuroPLC_Weights".w0, lut_table := lut_tmp);
    // φ[22→4]: evaluate LUT (table offset 2010)
    FOR k := 0 TO 14 DO
        lut_tmp[k] := "NeuroPLC_Weights".w1[2010 + k];
    END_FOR;
    v3[4, 22] := "BsplineEval"(x := v0[22], lut_grid := "NeuroPLC_Weights".w0, lut_table := lut_tmp);
    // φ[23→4]: evaluate LUT (table offset 2025)
    FOR k := 0 TO 14 DO
        lut_tmp[k] := "NeuroPLC_Weights".w1[2025 + k];
    END_FOR;
    v3[4, 23] := "BsplineEval"(x := v0[23], lut_grid := "NeuroPLC_Weights".w0, lut_table := lut_tmp);
    // φ[24→4]: evaluate LUT (table offset 2040)
    FOR k := 0 TO 14 DO
        lut_tmp[k] := "NeuroPLC_Weights".w1[2040 + k];
    END_FOR;
    v3[4, 24] := "BsplineEval"(x := v0[24], lut_grid := "NeuroPLC_Weights".w0, lut_table := lut_tmp);
    // φ[25→4]: evaluate LUT (table offset 2055)
    FOR k := 0 TO 14 DO
        lut_tmp[k] := "NeuroPLC_Weights".w1[2055 + k];
    END_FOR;
    v3[4, 25] := "BsplineEval"(x := v0[25], lut_grid := "NeuroPLC_Weights".w0, lut_table := lut_tmp);
    // φ[26→4]: evaluate LUT (table offset 2070)
    FOR k := 0 TO 14 DO
        lut_tmp[k] := "NeuroPLC_Weights".w1[2070 + k];
    END_FOR;
    v3[4, 26] := "BsplineEval"(x := v0[26], lut_grid := "NeuroPLC_Weights".w0, lut_table := lut_tmp);
    // φ[27→4]: evaluate LUT (table offset 2085)
    FOR k := 0 TO 14 DO
        lut_tmp[k] := "NeuroPLC_Weights".w1[2085 + k];
    END_FOR;
    v3[4, 27] := "BsplineEval"(x := v0[27], lut_grid := "NeuroPLC_Weights".w0, lut_table := lut_tmp);
    // φ[0→5]: evaluate LUT (table offset 2100)
    FOR k := 0 TO 14 DO
        lut_tmp[k] := "NeuroPLC_Weights".w1[2100 + k];
    END_FOR;
    v3[5, 0] := "BsplineEval"(x := v0[0], lut_grid := "NeuroPLC_Weights".w0, lut_table := lut_tmp);
    // φ[1→5]: evaluate LUT (table offset 2115)
    FOR k := 0 TO 14 DO
        lut_tmp[k] := "NeuroPLC_Weights".w1[2115 + k];
    END_FOR;
    v3[5, 1] := "BsplineEval"(x := v0[1], lut_grid := "NeuroPLC_Weights".w0, lut_table := lut_tmp);
    // φ[2→5]: evaluate LUT (table offset 2130)
    FOR k := 0 TO 14 DO
        lut_tmp[k] := "NeuroPLC_Weights".w1[2130 + k];
    END_FOR;
    v3[5, 2] := "BsplineEval"(x := v0[2], lut_grid := "NeuroPLC_Weights".w0, lut_table := lut_tmp);
    // φ[3→5]: evaluate LUT (table offset 2145)
    FOR k := 0 TO 14 DO
        lut_tmp[k] := "NeuroPLC_Weights".w1[2145 + k];
    END_FOR;
    v3[5, 3] := "BsplineEval"(x := v0[3], lut_grid := "NeuroPLC_Weights".w0, lut_table := lut_tmp);
    // φ[4→5]: evaluate LUT (table offset 2160)
    FOR k := 0 TO 14 DO
        lut_tmp[k] := "NeuroPLC_Weights".w1[2160 + k];
    END_FOR;
    v3[5, 4] := "BsplineEval"(x := v0[4], lut_grid := "NeuroPLC_Weights".w0, lut_table := lut_tmp);
    // φ[5→5]: evaluate LUT (table offset 2175)
    FOR k := 0 TO 14 DO
        lut_tmp[k] := "NeuroPLC_Weights".w1[2175 + k];
    END_FOR;
    v3[5, 5] := "BsplineEval"(x := v0[5], lut_grid := "NeuroPLC_Weights".w0, lut_table := lut_tmp);
    // φ[6→5]: evaluate LUT (table offset 2190)
    FOR k := 0 TO 14 DO
        lut_tmp[k] := "NeuroPLC_Weights".w1[2190 + k];
    END_FOR;
    v3[5, 6] := "BsplineEval"(x := v0[6], lut_grid := "NeuroPLC_Weights".w0, lut_table := lut_tmp);
    // φ[7→5]: evaluate LUT (table offset 2205)
    FOR k := 0 TO 14 DO
        lut_tmp[k] := "NeuroPLC_Weights".w1[2205 + k];
    END_FOR;
    v3[5, 7] := "BsplineEval"(x := v0[7], lut_grid := "NeuroPLC_Weights".w0, lut_table := lut_tmp);
    // φ[8→5]: evaluate LUT (table offset 2220)
    FOR k := 0 TO 14 DO
        lut_tmp[k] := "NeuroPLC_Weights".w1[2220 + k];
    END_FOR;
    v3[5, 8] := "BsplineEval"(x := v0[8], lut_grid := "NeuroPLC_Weights".w0, lut_table := lut_tmp);
    // φ[9→5]: evaluate LUT (table offset 2235)
    FOR k := 0 TO 14 DO
        lut_tmp[k] := "NeuroPLC_Weights".w1[2235 + k];
    END_FOR;
    v3[5, 9] := "BsplineEval"(x := v0[9], lut_grid := "NeuroPLC_Weights".w0, lut_table := lut_tmp);
    // φ[10→5]: evaluate LUT (table offset 2250)
    FOR k := 0 TO 14 DO
        lut_tmp[k] := "NeuroPLC_Weights".w1[2250 + k];
    END_FOR;
    v3[5, 10] := "BsplineEval"(x := v0[10], lut_grid := "NeuroPLC_Weights".w0, lut_table := lut_tmp);
    // φ[11→5]: evaluate LUT (table offset 2265)
    FOR k := 0 TO 14 DO
        lut_tmp[k] := "NeuroPLC_Weights".w1[2265 + k];
    END_FOR;
    v3[5, 11] := "BsplineEval"(x := v0[11], lut_grid := "NeuroPLC_Weights".w0, lut_table := lut_tmp);
    // φ[12→5]: evaluate LUT (table offset 2280)
    FOR k := 0 TO 14 DO
        lut_tmp[k] := "NeuroPLC_Weights".w1[2280 + k];
    END_FOR;
    v3[5, 12] := "BsplineEval"(x := v0[12], lut_grid := "NeuroPLC_Weights".w0, lut_table := lut_tmp);
    // φ[13→5]: evaluate LUT (table offset 2295)
    FOR k := 0 TO 14 DO
        lut_tmp[k] := "NeuroPLC_Weights".w1[2295 + k];
    END_FOR;
    v3[5, 13] := "BsplineEval"(x := v0[13], lut_grid := "NeuroPLC_Weights".w0, lut_table := lut_tmp);
    // φ[14→5]: evaluate LUT (table offset 2310)
    FOR k := 0 TO 14 DO
        lut_tmp[k] := "NeuroPLC_Weights".w1[2310 + k];
    END_FOR;
    v3[5, 14] := "BsplineEval"(x := v0[14], lut_grid := "NeuroPLC_Weights".w0, lut_table := lut_tmp);
    // φ[15→5]: evaluate LUT (table offset 2325)
    FOR k := 0 TO 14 DO
        lut_tmp[k] := "NeuroPLC_Weights".w1[2325 + k];
    END_FOR;
    v3[5, 15] := "BsplineEval"(x := v0[15], lut_grid := "NeuroPLC_Weights".w0, lut_table := lut_tmp);
    // φ[16→5]: evaluate LUT (table offset 2340)
    FOR k := 0 TO 14 DO
        lut_tmp[k] := "NeuroPLC_Weights".w1[2340 + k];
    END_FOR;
    v3[5, 16] := "BsplineEval"(x := v0[16], lut_grid := "NeuroPLC_Weights".w0, lut_table := lut_tmp);
    // φ[17→5]: evaluate LUT (table offset 2355)
    FOR k := 0 TO 14 DO
        lut_tmp[k] := "NeuroPLC_Weights".w1[2355 + k];
    END_FOR;
    v3[5, 17] := "BsplineEval"(x := v0[17], lut_grid := "NeuroPLC_Weights".w0, lut_table := lut_tmp);
    // φ[18→5]: evaluate LUT (table offset 2370)
    FOR k := 0 TO 14 DO
        lut_tmp[k] := "NeuroPLC_Weights".w1[2370 + k];
    END_FOR;
    v3[5, 18] := "BsplineEval"(x := v0[18], lut_grid := "NeuroPLC_Weights".w0, lut_table := lut_tmp);
    // φ[19→5]: evaluate LUT (table offset 2385)
    FOR k := 0 TO 14 DO
        lut_tmp[k] := "NeuroPLC_Weights".w1[2385 + k];
    END_FOR;
    v3[5, 19] := "BsplineEval"(x := v0[19], lut_grid := "NeuroPLC_Weights".w0, lut_table := lut_tmp);
    // φ[20→5]: evaluate LUT (table offset 2400)
    FOR k := 0 TO 14 DO
        lut_tmp[k] := "NeuroPLC_Weights".w1[2400 + k];
    END_FOR;
    v3[5, 20] := "BsplineEval"(x := v0[20], lut_grid := "NeuroPLC_Weights".w0, lut_table := lut_tmp);
    // φ[21→5]: evaluate LUT (table offset 2415)
    FOR k := 0 TO 14 DO
        lut_tmp[k] := "NeuroPLC_Weights".w1[2415 + k];
    END_FOR;
    v3[5, 21] := "BsplineEval"(x := v0[21], lut_grid := "NeuroPLC_Weights".w0, lut_table := lut_tmp);
    // φ[22→5]: evaluate LUT (table offset 2430)
    FOR k := 0 TO 14 DO
        lut_tmp[k] := "NeuroPLC_Weights".w1[2430 + k];
    END_FOR;
    v3[5, 22] := "BsplineEval"(x := v0[22], lut_grid := "NeuroPLC_Weights".w0, lut_table := lut_tmp);
    // φ[23→5]: evaluate LUT (table offset 2445)
    FOR k := 0 TO 14 DO
        lut_tmp[k] := "NeuroPLC_Weights".w1[2445 + k];
    END_FOR;
    v3[5, 23] := "BsplineEval"(x := v0[23], lut_grid := "NeuroPLC_Weights".w0, lut_table := lut_tmp);
    // φ[24→5]: evaluate LUT (table offset 2460)
    FOR k := 0 TO 14 DO
        lut_tmp[k] := "NeuroPLC_Weights".w1[2460 + k];
    END_FOR;
    v3[5, 24] := "BsplineEval"(x := v0[24], lut_grid := "NeuroPLC_Weights".w0, lut_table := lut_tmp);
    // φ[25→5]: evaluate LUT (table offset 2475)
    FOR k := 0 TO 14 DO
        lut_tmp[k] := "NeuroPLC_Weights".w1[2475 + k];
    END_FOR;
    v3[5, 25] := "BsplineEval"(x := v0[25], lut_grid := "NeuroPLC_Weights".w0, lut_table := lut_tmp);
    // φ[26→5]: evaluate LUT (table offset 2490)
    FOR k := 0 TO 14 DO
        lut_tmp[k] := "NeuroPLC_Weights".w1[2490 + k];
    END_FOR;
    v3[5, 26] := "BsplineEval"(x := v0[26], lut_grid := "NeuroPLC_Weights".w0, lut_table := lut_tmp);
    // φ[27→5]: evaluate LUT (table offset 2505)
    FOR k := 0 TO 14 DO
        lut_tmp[k] := "NeuroPLC_Weights".w1[2505 + k];
    END_FOR;
    v3[5, 27] := "BsplineEval"(x := v0[27], lut_grid := "NeuroPLC_Weights".w0, lut_table := lut_tmp);
    // φ[0→6]: evaluate LUT (table offset 2520)
    FOR k := 0 TO 14 DO
        lut_tmp[k] := "NeuroPLC_Weights".w1[2520 + k];
    END_FOR;
    v3[6, 0] := "BsplineEval"(x := v0[0], lut_grid := "NeuroPLC_Weights".w0, lut_table := lut_tmp);
    // φ[1→6]: evaluate LUT (table offset 2535)
    FOR k := 0 TO 14 DO
        lut_tmp[k] := "NeuroPLC_Weights".w1[2535 + k];
    END_FOR;
    v3[6, 1] := "BsplineEval"(x := v0[1], lut_grid := "NeuroPLC_Weights".w0, lut_table := lut_tmp);
    // φ[2→6]: evaluate LUT (table offset 2550)
    FOR k := 0 TO 14 DO
        lut_tmp[k] := "NeuroPLC_Weights".w1[2550 + k];
    END_FOR;
    v3[6, 2] := "BsplineEval"(x := v0[2], lut_grid := "NeuroPLC_Weights".w0, lut_table := lut_tmp);
    // φ[3→6]: evaluate LUT (table offset 2565)
    FOR k := 0 TO 14 DO
        lut_tmp[k] := "NeuroPLC_Weights".w1[2565 + k];
    END_FOR;
    v3[6, 3] := "BsplineEval"(x := v0[3], lut_grid := "NeuroPLC_Weights".w0, lut_table := lut_tmp);
    // φ[4→6]: evaluate LUT (table offset 2580)
    FOR k := 0 TO 14 DO
        lut_tmp[k] := "NeuroPLC_Weights".w1[2580 + k];
    END_FOR;
    v3[6, 4] := "BsplineEval"(x := v0[4], lut_grid := "NeuroPLC_Weights".w0, lut_table := lut_tmp);
    // φ[5→6]: evaluate LUT (table offset 2595)
    FOR k := 0 TO 14 DO
        lut_tmp[k] := "NeuroPLC_Weights".w1[2595 + k];
    END_FOR;
    v3[6, 5] := "BsplineEval"(x := v0[5], lut_grid := "NeuroPLC_Weights".w0, lut_table := lut_tmp);
    // φ[6→6]: evaluate LUT (table offset 2610)
    FOR k := 0 TO 14 DO
        lut_tmp[k] := "NeuroPLC_Weights".w1[2610 + k];
    END_FOR;
    v3[6, 6] := "BsplineEval"(x := v0[6], lut_grid := "NeuroPLC_Weights".w0, lut_table := lut_tmp);
    // φ[7→6]: evaluate LUT (table offset 2625)
    FOR k := 0 TO 14 DO
        lut_tmp[k] := "NeuroPLC_Weights".w1[2625 + k];
    END_FOR;
    v3[6, 7] := "BsplineEval"(x := v0[7], lut_grid := "NeuroPLC_Weights".w0, lut_table := lut_tmp);
    // φ[8→6]: evaluate LUT (table offset 2640)
    FOR k := 0 TO 14 DO
        lut_tmp[k] := "NeuroPLC_Weights".w1[2640 + k];
    END_FOR;
    v3[6, 8] := "BsplineEval"(x := v0[8], lut_grid := "NeuroPLC_Weights".w0, lut_table := lut_tmp);
    // φ[9→6]: evaluate LUT (table offset 2655)
    FOR k := 0 TO 14 DO
        lut_tmp[k] := "NeuroPLC_Weights".w1[2655 + k];
    END_FOR;
    v3[6, 9] := "BsplineEval"(x := v0[9], lut_grid := "NeuroPLC_Weights".w0, lut_table := lut_tmp);
    // φ[10→6]: evaluate LUT (table offset 2670)
    FOR k := 0 TO 14 DO
        lut_tmp[k] := "NeuroPLC_Weights".w1[2670 + k];
    END_FOR;
    v3[6, 10] := "BsplineEval"(x := v0[10], lut_grid := "NeuroPLC_Weights".w0, lut_table := lut_tmp);
    // φ[11→6]: evaluate LUT (table offset 2685)
    FOR k := 0 TO 14 DO
        lut_tmp[k] := "NeuroPLC_Weights".w1[2685 + k];
    END_FOR;
    v3[6, 11] := "BsplineEval"(x := v0[11], lut_grid := "NeuroPLC_Weights".w0, lut_table := lut_tmp);
    // φ[12→6]: evaluate LUT (table offset 2700)
    FOR k := 0 TO 14 DO
        lut_tmp[k] := "NeuroPLC_Weights".w1[2700 + k];
    END_FOR;
    v3[6, 12] := "BsplineEval"(x := v0[12], lut_grid := "NeuroPLC_Weights".w0, lut_table := lut_tmp);
    // φ[13→6]: evaluate LUT (table offset 2715)
    FOR k := 0 TO 14 DO
        lut_tmp[k] := "NeuroPLC_Weights".w1[2715 + k];
    END_FOR;
    v3[6, 13] := "BsplineEval"(x := v0[13], lut_grid := "NeuroPLC_Weights".w0, lut_table := lut_tmp);
    // φ[14→6]: evaluate LUT (table offset 2730)
    FOR k := 0 TO 14 DO
        lut_tmp[k] := "NeuroPLC_Weights".w1[2730 + k];
    END_FOR;
    v3[6, 14] := "BsplineEval"(x := v0[14], lut_grid := "NeuroPLC_Weights".w0, lut_table := lut_tmp);
    // φ[15→6]: evaluate LUT (table offset 2745)
    FOR k := 0 TO 14 DO
        lut_tmp[k] := "NeuroPLC_Weights".w1[2745 + k];
    END_FOR;
    v3[6, 15] := "BsplineEval"(x := v0[15], lut_grid := "NeuroPLC_Weights".w0, lut_table := lut_tmp);
    // φ[16→6]: evaluate LUT (table offset 2760)
    FOR k := 0 TO 14 DO
        lut_tmp[k] := "NeuroPLC_Weights".w1[2760 + k];
    END_FOR;
    v3[6, 16] := "BsplineEval"(x := v0[16], lut_grid := "NeuroPLC_Weights".w0, lut_table := lut_tmp);
    // φ[17→6]: evaluate LUT (table offset 2775)
    FOR k := 0 TO 14 DO
        lut_tmp[k] := "NeuroPLC_Weights".w1[2775 + k];
    END_FOR;
    v3[6, 17] := "BsplineEval"(x := v0[17], lut_grid := "NeuroPLC_Weights".w0, lut_table := lut_tmp);
    // φ[18→6]: evaluate LUT (table offset 2790)
    FOR k := 0 TO 14 DO
        lut_tmp[k] := "NeuroPLC_Weights".w1[2790 + k];
    END_FOR;
    v3[6, 18] := "BsplineEval"(x := v0[18], lut_grid := "NeuroPLC_Weights".w0, lut_table := lut_tmp);
    // φ[19→6]: evaluate LUT (table offset 2805)
    FOR k := 0 TO 14 DO
        lut_tmp[k] := "NeuroPLC_Weights".w1[2805 + k];
    END_FOR;
    v3[6, 19] := "BsplineEval"(x := v0[19], lut_grid := "NeuroPLC_Weights".w0, lut_table := lut_tmp);
    // φ[20→6]: evaluate LUT (table offset 2820)
    FOR k := 0 TO 14 DO
        lut_tmp[k] := "NeuroPLC_Weights".w1[2820 + k];
    END_FOR;
    v3[6, 20] := "BsplineEval"(x := v0[20], lut_grid := "NeuroPLC_Weights".w0, lut_table := lut_tmp);
    // φ[21→6]: evaluate LUT (table offset 2835)
    FOR k := 0 TO 14 DO
        lut_tmp[k] := "NeuroPLC_Weights".w1[2835 + k];
    END_FOR;
    v3[6, 21] := "BsplineEval"(x := v0[21], lut_grid := "NeuroPLC_Weights".w0, lut_table := lut_tmp);
    // φ[22→6]: evaluate LUT (table offset 2850)
    FOR k := 0 TO 14 DO
        lut_tmp[k] := "NeuroPLC_Weights".w1[2850 + k];
    END_FOR;
    v3[6, 22] := "BsplineEval"(x := v0[22], lut_grid := "NeuroPLC_Weights".w0, lut_table := lut_tmp);
    // φ[23→6]: evaluate LUT (table offset 2865)
    FOR k := 0 TO 14 DO
        lut_tmp[k] := "NeuroPLC_Weights".w1[2865 + k];
    END_FOR;
    v3[6, 23] := "BsplineEval"(x := v0[23], lut_grid := "NeuroPLC_Weights".w0, lut_table := lut_tmp);
    // φ[24→6]: evaluate LUT (table offset 2880)
    FOR k := 0 TO 14 DO
        lut_tmp[k] := "NeuroPLC_Weights".w1[2880 + k];
    END_FOR;
    v3[6, 24] := "BsplineEval"(x := v0[24], lut_grid := "NeuroPLC_Weights".w0, lut_table := lut_tmp);
    // φ[25→6]: evaluate LUT (table offset 2895)
    FOR k := 0 TO 14 DO
        lut_tmp[k] := "NeuroPLC_Weights".w1[2895 + k];
    END_FOR;
    v3[6, 25] := "BsplineEval"(x := v0[25], lut_grid := "NeuroPLC_Weights".w0, lut_table := lut_tmp);
    // φ[26→6]: evaluate LUT (table offset 2910)
    FOR k := 0 TO 14 DO
        lut_tmp[k] := "NeuroPLC_Weights".w1[2910 + k];
    END_FOR;
    v3[6, 26] := "BsplineEval"(x := v0[26], lut_grid := "NeuroPLC_Weights".w0, lut_table := lut_tmp);
    // φ[27→6]: evaluate LUT (table offset 2925)
    FOR k := 0 TO 14 DO
        lut_tmp[k] := "NeuroPLC_Weights".w1[2925 + k];
    END_FOR;
    v3[6, 27] := "BsplineEval"(x := v0[27], lut_grid := "NeuroPLC_Weights".w0, lut_table := lut_tmp);
    // φ[0→7]: evaluate LUT (table offset 2940)
    FOR k := 0 TO 14 DO
        lut_tmp[k] := "NeuroPLC_Weights".w1[2940 + k];
    END_FOR;
    v3[7, 0] := "BsplineEval"(x := v0[0], lut_grid := "NeuroPLC_Weights".w0, lut_table := lut_tmp);
    // φ[1→7]: evaluate LUT (table offset 2955)
    FOR k := 0 TO 14 DO
        lut_tmp[k] := "NeuroPLC_Weights".w1[2955 + k];
    END_FOR;
    v3[7, 1] := "BsplineEval"(x := v0[1], lut_grid := "NeuroPLC_Weights".w0, lut_table := lut_tmp);
    // φ[2→7]: evaluate LUT (table offset 2970)
    FOR k := 0 TO 14 DO
        lut_tmp[k] := "NeuroPLC_Weights".w1[2970 + k];
    END_FOR;
    v3[7, 2] := "BsplineEval"(x := v0[2], lut_grid := "NeuroPLC_Weights".w0, lut_table := lut_tmp);
    // φ[3→7]: evaluate LUT (table offset 2985)
    FOR k := 0 TO 14 DO
        lut_tmp[k] := "NeuroPLC_Weights".w1[2985 + k];
    END_FOR;
    v3[7, 3] := "BsplineEval"(x := v0[3], lut_grid := "NeuroPLC_Weights".w0, lut_table := lut_tmp);
    // φ[4→7]: evaluate LUT (table offset 3000)
    FOR k := 0 TO 14 DO
        lut_tmp[k] := "NeuroPLC_Weights".w1[3000 + k];
    END_FOR;
    v3[7, 4] := "BsplineEval"(x := v0[4], lut_grid := "NeuroPLC_Weights".w0, lut_table := lut_tmp);
    // φ[5→7]: evaluate LUT (table offset 3015)
    FOR k := 0 TO 14 DO
        lut_tmp[k] := "NeuroPLC_Weights".w1[3015 + k];
    END_FOR;
    v3[7, 5] := "BsplineEval"(x := v0[5], lut_grid := "NeuroPLC_Weights".w0, lut_table := lut_tmp);
    // φ[6→7]: evaluate LUT (table offset 3030)
    FOR k := 0 TO 14 DO
        lut_tmp[k] := "NeuroPLC_Weights".w1[3030 + k];
    END_FOR;
    v3[7, 6] := "BsplineEval"(x := v0[6], lut_grid := "NeuroPLC_Weights".w0, lut_table := lut_tmp);
    // φ[7→7]: evaluate LUT (table offset 3045)
    FOR k := 0 TO 14 DO
        lut_tmp[k] := "NeuroPLC_Weights".w1[3045 + k];
    END_FOR;
    v3[7, 7] := "BsplineEval"(x := v0[7], lut_grid := "NeuroPLC_Weights".w0, lut_table := lut_tmp);
    // φ[8→7]: evaluate LUT (table offset 3060)
    FOR k := 0 TO 14 DO
        lut_tmp[k] := "NeuroPLC_Weights".w1[3060 + k];
    END_FOR;
    v3[7, 8] := "BsplineEval"(x := v0[8], lut_grid := "NeuroPLC_Weights".w0, lut_table := lut_tmp);
    // φ[9→7]: evaluate LUT (table offset 3075)
    FOR k := 0 TO 14 DO
        lut_tmp[k] := "NeuroPLC_Weights".w1[3075 + k];
    END_FOR;
    v3[7, 9] := "BsplineEval"(x := v0[9], lut_grid := "NeuroPLC_Weights".w0, lut_table := lut_tmp);
    // φ[10→7]: evaluate LUT (table offset 3090)
    FOR k := 0 TO 14 DO
        lut_tmp[k] := "NeuroPLC_Weights".w1[3090 + k];
    END_FOR;
    v3[7, 10] := "BsplineEval"(x := v0[10], lut_grid := "NeuroPLC_Weights".w0, lut_table := lut_tmp);
    // φ[11→7]: evaluate LUT (table offset 3105)
    FOR k := 0 TO 14 DO
        lut_tmp[k] := "NeuroPLC_Weights".w1[3105 + k];
    END_FOR;
    v3[7, 11] := "BsplineEval"(x := v0[11], lut_grid := "NeuroPLC_Weights".w0, lut_table := lut_tmp);
    // φ[12→7]: evaluate LUT (table offset 3120)
    FOR k := 0 TO 14 DO
        lut_tmp[k] := "NeuroPLC_Weights".w1[3120 + k];
    END_FOR;
    v3[7, 12] := "BsplineEval"(x := v0[12], lut_grid := "NeuroPLC_Weights".w0, lut_table := lut_tmp);
    // φ[13→7]: evaluate LUT (table offset 3135)
    FOR k := 0 TO 14 DO
        lut_tmp[k] := "NeuroPLC_Weights".w1[3135 + k];
    END_FOR;
    v3[7, 13] := "BsplineEval"(x := v0[13], lut_grid := "NeuroPLC_Weights".w0, lut_table := lut_tmp);
    // φ[14→7]: evaluate LUT (table offset 3150)
    FOR k := 0 TO 14 DO
        lut_tmp[k] := "NeuroPLC_Weights".w1[3150 + k];
    END_FOR;
    v3[7, 14] := "BsplineEval"(x := v0[14], lut_grid := "NeuroPLC_Weights".w0, lut_table := lut_tmp);
    // φ[15→7]: evaluate LUT (table offset 3165)
    FOR k := 0 TO 14 DO
        lut_tmp[k] := "NeuroPLC_Weights".w1[3165 + k];
    END_FOR;
    v3[7, 15] := "BsplineEval"(x := v0[15], lut_grid := "NeuroPLC_Weights".w0, lut_table := lut_tmp);
    // φ[16→7]: evaluate LUT (table offset 3180)
    FOR k := 0 TO 14 DO
        lut_tmp[k] := "NeuroPLC_Weights".w1[3180 + k];
    END_FOR;
    v3[7, 16] := "BsplineEval"(x := v0[16], lut_grid := "NeuroPLC_Weights".w0, lut_table := lut_tmp);
    // φ[17→7]: evaluate LUT (table offset 3195)
    FOR k := 0 TO 14 DO
        lut_tmp[k] := "NeuroPLC_Weights".w1[3195 + k];
    END_FOR;
    v3[7, 17] := "BsplineEval"(x := v0[17], lut_grid := "NeuroPLC_Weights".w0, lut_table := lut_tmp);
    // φ[18→7]: evaluate LUT (table offset 3210)
    FOR k := 0 TO 14 DO
        lut_tmp[k] := "NeuroPLC_Weights".w1[3210 + k];
    END_FOR;
    v3[7, 18] := "BsplineEval"(x := v0[18], lut_grid := "NeuroPLC_Weights".w0, lut_table := lut_tmp);
    // φ[19→7]: evaluate LUT (table offset 3225)
    FOR k := 0 TO 14 DO
        lut_tmp[k] := "NeuroPLC_Weights".w1[3225 + k];
    END_FOR;
    v3[7, 19] := "BsplineEval"(x := v0[19], lut_grid := "NeuroPLC_Weights".w0, lut_table := lut_tmp);
    // φ[20→7]: evaluate LUT (table offset 3240)
    FOR k := 0 TO 14 DO
        lut_tmp[k] := "NeuroPLC_Weights".w1[3240 + k];
    END_FOR;
    v3[7, 20] := "BsplineEval"(x := v0[20], lut_grid := "NeuroPLC_Weights".w0, lut_table := lut_tmp);
    // φ[21→7]: evaluate LUT (table offset 3255)
    FOR k := 0 TO 14 DO
        lut_tmp[k] := "NeuroPLC_Weights".w1[3255 + k];
    END_FOR;
    v3[7, 21] := "BsplineEval"(x := v0[21], lut_grid := "NeuroPLC_Weights".w0, lut_table := lut_tmp);
    // φ[22→7]: evaluate LUT (table offset 3270)
    FOR k := 0 TO 14 DO
        lut_tmp[k] := "NeuroPLC_Weights".w1[3270 + k];
    END_FOR;
    v3[7, 22] := "BsplineEval"(x := v0[22], lut_grid := "NeuroPLC_Weights".w0, lut_table := lut_tmp);
    // φ[23→7]: evaluate LUT (table offset 3285)
    FOR k := 0 TO 14 DO
        lut_tmp[k] := "NeuroPLC_Weights".w1[3285 + k];
    END_FOR;
    v3[7, 23] := "BsplineEval"(x := v0[23], lut_grid := "NeuroPLC_Weights".w0, lut_table := lut_tmp);
    // φ[24→7]: evaluate LUT (table offset 3300)
    FOR k := 0 TO 14 DO
        lut_tmp[k] := "NeuroPLC_Weights".w1[3300 + k];
    END_FOR;
    v3[7, 24] := "BsplineEval"(x := v0[24], lut_grid := "NeuroPLC_Weights".w0, lut_table := lut_tmp);
    // φ[25→7]: evaluate LUT (table offset 3315)
    FOR k := 0 TO 14 DO
        lut_tmp[k] := "NeuroPLC_Weights".w1[3315 + k];
    END_FOR;
    v3[7, 25] := "BsplineEval"(x := v0[25], lut_grid := "NeuroPLC_Weights".w0, lut_table := lut_tmp);
    // φ[26→7]: evaluate LUT (table offset 3330)
    FOR k := 0 TO 14 DO
        lut_tmp[k] := "NeuroPLC_Weights".w1[3330 + k];
    END_FOR;
    v3[7, 26] := "BsplineEval"(x := v0[26], lut_grid := "NeuroPLC_Weights".w0, lut_table := lut_tmp);
    // φ[27→7]: evaluate LUT (table offset 3345)
    FOR k := 0 TO 14 DO
        lut_tmp[k] := "NeuroPLC_Weights".w1[3345 + k];
    END_FOR;
    v3[7, 27] := "BsplineEval"(x := v0[27], lut_grid := "NeuroPLC_Weights".w0, lut_table := lut_tmp);
    // φ[0→8]: evaluate LUT (table offset 3360)
    FOR k := 0 TO 14 DO
        lut_tmp[k] := "NeuroPLC_Weights".w1[3360 + k];
    END_FOR;
    v3[8, 0] := "BsplineEval"(x := v0[0], lut_grid := "NeuroPLC_Weights".w0, lut_table := lut_tmp);
    // φ[1→8]: evaluate LUT (table offset 3375)
    FOR k := 0 TO 14 DO
        lut_tmp[k] := "NeuroPLC_Weights".w1[3375 + k];
    END_FOR;
    v3[8, 1] := "BsplineEval"(x := v0[1], lut_grid := "NeuroPLC_Weights".w0, lut_table := lut_tmp);
    // φ[2→8]: evaluate LUT (table offset 3390)
    FOR k := 0 TO 14 DO
        lut_tmp[k] := "NeuroPLC_Weights".w1[3390 + k];
    END_FOR;
    v3[8, 2] := "BsplineEval"(x := v0[2], lut_grid := "NeuroPLC_Weights".w0, lut_table := lut_tmp);
    // φ[3→8]: evaluate LUT (table offset 3405)
    FOR k := 0 TO 14 DO
        lut_tmp[k] := "NeuroPLC_Weights".w1[3405 + k];
    END_FOR;
    v3[8, 3] := "BsplineEval"(x := v0[3], lut_grid := "NeuroPLC_Weights".w0, lut_table := lut_tmp);
    // φ[4→8]: evaluate LUT (table offset 3420)
    FOR k := 0 TO 14 DO
        lut_tmp[k] := "NeuroPLC_Weights".w1[3420 + k];
    END_FOR;
    v3[8, 4] := "BsplineEval"(x := v0[4], lut_grid := "NeuroPLC_Weights".w0, lut_table := lut_tmp);
    // φ[5→8]: evaluate LUT (table offset 3435)
    FOR k := 0 TO 14 DO
        lut_tmp[k] := "NeuroPLC_Weights".w1[3435 + k];
    END_FOR;
    v3[8, 5] := "BsplineEval"(x := v0[5], lut_grid := "NeuroPLC_Weights".w0, lut_table := lut_tmp);
    // φ[6→8]: evaluate LUT (table offset 3450)
    FOR k := 0 TO 14 DO
        lut_tmp[k] := "NeuroPLC_Weights".w1[3450 + k];
    END_FOR;
    v3[8, 6] := "BsplineEval"(x := v0[6], lut_grid := "NeuroPLC_Weights".w0, lut_table := lut_tmp);
    // φ[7→8]: evaluate LUT (table offset 3465)
    FOR k := 0 TO 14 DO
        lut_tmp[k] := "NeuroPLC_Weights".w1[3465 + k];
    END_FOR;
    v3[8, 7] := "BsplineEval"(x := v0[7], lut_grid := "NeuroPLC_Weights".w0, lut_table := lut_tmp);
    // φ[8→8]: evaluate LUT (table offset 3480)
    FOR k := 0 TO 14 DO
        lut_tmp[k] := "NeuroPLC_Weights".w1[3480 + k];
    END_FOR;
    v3[8, 8] := "BsplineEval"(x := v0[8], lut_grid := "NeuroPLC_Weights".w0, lut_table := lut_tmp);
    // φ[9→8]: evaluate LUT (table offset 3495)
    FOR k := 0 TO 14 DO
        lut_tmp[k] := "NeuroPLC_Weights".w1[3495 + k];
    END_FOR;
    v3[8, 9] := "BsplineEval"(x := v0[9], lut_grid := "NeuroPLC_Weights".w0, lut_table := lut_tmp);
    // φ[10→8]: evaluate LUT (table offset 3510)
    FOR k := 0 TO 14 DO
        lut_tmp[k] := "NeuroPLC_Weights".w1[3510 + k];
    END_FOR;
    v3[8, 10] := "BsplineEval"(x := v0[10], lut_grid := "NeuroPLC_Weights".w0, lut_table := lut_tmp);
    // φ[11→8]: evaluate LUT (table offset 3525)
    FOR k := 0 TO 14 DO
        lut_tmp[k] := "NeuroPLC_Weights".w1[3525 + k];
    END_FOR;
    v3[8, 11] := "BsplineEval"(x := v0[11], lut_grid := "NeuroPLC_Weights".w0, lut_table := lut_tmp);
    // φ[12→8]: evaluate LUT (table offset 3540)
    FOR k := 0 TO 14 DO
        lut_tmp[k] := "NeuroPLC_Weights".w1[3540 + k];
    END_FOR;
    v3[8, 12] := "BsplineEval"(x := v0[12], lut_grid := "NeuroPLC_Weights".w0, lut_table := lut_tmp);
    // φ[13→8]: evaluate LUT (table offset 3555)
    FOR k := 0 TO 14 DO
        lut_tmp[k] := "NeuroPLC_Weights".w1[3555 + k];
    END_FOR;
    v3[8, 13] := "BsplineEval"(x := v0[13], lut_grid := "NeuroPLC_Weights".w0, lut_table := lut_tmp);
    // φ[14→8]: evaluate LUT (table offset 3570)
    FOR k := 0 TO 14 DO
        lut_tmp[k] := "NeuroPLC_Weights".w1[3570 + k];
    END_FOR;
    v3[8, 14] := "BsplineEval"(x := v0[14], lut_grid := "NeuroPLC_Weights".w0, lut_table := lut_tmp);
    // φ[15→8]: evaluate LUT (table offset 3585)
    FOR k := 0 TO 14 DO
        lut_tmp[k] := "NeuroPLC_Weights".w1[3585 + k];
    END_FOR;
    v3[8, 15] := "BsplineEval"(x := v0[15], lut_grid := "NeuroPLC_Weights".w0, lut_table := lut_tmp);
    // φ[16→8]: evaluate LUT (table offset 3600)
    FOR k := 0 TO 14 DO
        lut_tmp[k] := "NeuroPLC_Weights".w1[3600 + k];
    END_FOR;
    v3[8, 16] := "BsplineEval"(x := v0[16], lut_grid := "NeuroPLC_Weights".w0, lut_table := lut_tmp);
    // φ[17→8]: evaluate LUT (table offset 3615)
    FOR k := 0 TO 14 DO
        lut_tmp[k] := "NeuroPLC_Weights".w1[3615 + k];
    END_FOR;
    v3[8, 17] := "BsplineEval"(x := v0[17], lut_grid := "NeuroPLC_Weights".w0, lut_table := lut_tmp);
    // φ[18→8]: evaluate LUT (table offset 3630)
    FOR k := 0 TO 14 DO
        lut_tmp[k] := "NeuroPLC_Weights".w1[3630 + k];
    END_FOR;
    v3[8, 18] := "BsplineEval"(x := v0[18], lut_grid := "NeuroPLC_Weights".w0, lut_table := lut_tmp);
    // φ[19→8]: evaluate LUT (table offset 3645)
    FOR k := 0 TO 14 DO
        lut_tmp[k] := "NeuroPLC_Weights".w1[3645 + k];
    END_FOR;
    v3[8, 19] := "BsplineEval"(x := v0[19], lut_grid := "NeuroPLC_Weights".w0, lut_table := lut_tmp);
    // φ[20→8]: evaluate LUT (table offset 3660)
    FOR k := 0 TO 14 DO
        lut_tmp[k] := "NeuroPLC_Weights".w1[3660 + k];
    END_FOR;
    v3[8, 20] := "BsplineEval"(x := v0[20], lut_grid := "NeuroPLC_Weights".w0, lut_table := lut_tmp);
    // φ[21→8]: evaluate LUT (table offset 3675)
    FOR k := 0 TO 14 DO
        lut_tmp[k] := "NeuroPLC_Weights".w1[3675 + k];
    END_FOR;
    v3[8, 21] := "BsplineEval"(x := v0[21], lut_grid := "NeuroPLC_Weights".w0, lut_table := lut_tmp);
    // φ[22→8]: evaluate LUT (table offset 3690)
    FOR k := 0 TO 14 DO
        lut_tmp[k] := "NeuroPLC_Weights".w1[3690 + k];
    END_FOR;
    v3[8, 22] := "BsplineEval"(x := v0[22], lut_grid := "NeuroPLC_Weights".w0, lut_table := lut_tmp);
    // φ[23→8]: evaluate LUT (table offset 3705)
    FOR k := 0 TO 14 DO
        lut_tmp[k] := "NeuroPLC_Weights".w1[3705 + k];
    END_FOR;
    v3[8, 23] := "BsplineEval"(x := v0[23], lut_grid := "NeuroPLC_Weights".w0, lut_table := lut_tmp);
    // φ[24→8]: evaluate LUT (table offset 3720)
    FOR k := 0 TO 14 DO
        lut_tmp[k] := "NeuroPLC_Weights".w1[3720 + k];
    END_FOR;
    v3[8, 24] := "BsplineEval"(x := v0[24], lut_grid := "NeuroPLC_Weights".w0, lut_table := lut_tmp);
    // φ[25→8]: evaluate LUT (table offset 3735)
    FOR k := 0 TO 14 DO
        lut_tmp[k] := "NeuroPLC_Weights".w1[3735 + k];
    END_FOR;
    v3[8, 25] := "BsplineEval"(x := v0[25], lut_grid := "NeuroPLC_Weights".w0, lut_table := lut_tmp);
    // φ[26→8]: evaluate LUT (table offset 3750)
    FOR k := 0 TO 14 DO
        lut_tmp[k] := "NeuroPLC_Weights".w1[3750 + k];
    END_FOR;
    v3[8, 26] := "BsplineEval"(x := v0[26], lut_grid := "NeuroPLC_Weights".w0, lut_table := lut_tmp);
    // φ[27→8]: evaluate LUT (table offset 3765)
    FOR k := 0 TO 14 DO
        lut_tmp[k] := "NeuroPLC_Weights".w1[3765 + k];
    END_FOR;
    v3[8, 27] := "BsplineEval"(x := v0[27], lut_grid := "NeuroPLC_Weights".w0, lut_table := lut_tmp);
    // φ[0→9]: evaluate LUT (table offset 3780)
    FOR k := 0 TO 14 DO
        lut_tmp[k] := "NeuroPLC_Weights".w1[3780 + k];
    END_FOR;
    v3[9, 0] := "BsplineEval"(x := v0[0], lut_grid := "NeuroPLC_Weights".w0, lut_table := lut_tmp);
    // φ[1→9]: evaluate LUT (table offset 3795)
    FOR k := 0 TO 14 DO
        lut_tmp[k] := "NeuroPLC_Weights".w1[3795 + k];
    END_FOR;
    v3[9, 1] := "BsplineEval"(x := v0[1], lut_grid := "NeuroPLC_Weights".w0, lut_table := lut_tmp);
    // φ[2→9]: evaluate LUT (table offset 3810)
    FOR k := 0 TO 14 DO
        lut_tmp[k] := "NeuroPLC_Weights".w1[3810 + k];
    END_FOR;
    v3[9, 2] := "BsplineEval"(x := v0[2], lut_grid := "NeuroPLC_Weights".w0, lut_table := lut_tmp);
    // φ[3→9]: evaluate LUT (table offset 3825)
    FOR k := 0 TO 14 DO
        lut_tmp[k] := "NeuroPLC_Weights".w1[3825 + k];
    END_FOR;
    v3[9, 3] := "BsplineEval"(x := v0[3], lut_grid := "NeuroPLC_Weights".w0, lut_table := lut_tmp);
    // φ[4→9]: evaluate LUT (table offset 3840)
    FOR k := 0 TO 14 DO
        lut_tmp[k] := "NeuroPLC_Weights".w1[3840 + k];
    END_FOR;
    v3[9, 4] := "BsplineEval"(x := v0[4], lut_grid := "NeuroPLC_Weights".w0, lut_table := lut_tmp);
    // φ[5→9]: evaluate LUT (table offset 3855)
    FOR k := 0 TO 14 DO
        lut_tmp[k] := "NeuroPLC_Weights".w1[3855 + k];
    END_FOR;
    v3[9, 5] := "BsplineEval"(x := v0[5], lut_grid := "NeuroPLC_Weights".w0, lut_table := lut_tmp);
    // φ[6→9]: evaluate LUT (table offset 3870)
    FOR k := 0 TO 14 DO
        lut_tmp[k] := "NeuroPLC_Weights".w1[3870 + k];
    END_FOR;
    v3[9, 6] := "BsplineEval"(x := v0[6], lut_grid := "NeuroPLC_Weights".w0, lut_table := lut_tmp);
    // φ[7→9]: evaluate LUT (table offset 3885)
    FOR k := 0 TO 14 DO
        lut_tmp[k] := "NeuroPLC_Weights".w1[3885 + k];
    END_FOR;
    v3[9, 7] := "BsplineEval"(x := v0[7], lut_grid := "NeuroPLC_Weights".w0, lut_table := lut_tmp);
    // φ[8→9]: evaluate LUT (table offset 3900)
    FOR k := 0 TO 14 DO
        lut_tmp[k] := "NeuroPLC_Weights".w1[3900 + k];
    END_FOR;
    v3[9, 8] := "BsplineEval"(x := v0[8], lut_grid := "NeuroPLC_Weights".w0, lut_table := lut_tmp);
    // φ[9→9]: evaluate LUT (table offset 3915)
    FOR k := 0 TO 14 DO
        lut_tmp[k] := "NeuroPLC_Weights".w1[3915 + k];
    END_FOR;
    v3[9, 9] := "BsplineEval"(x := v0[9], lut_grid := "NeuroPLC_Weights".w0, lut_table := lut_tmp);
    // φ[10→9]: evaluate LUT (table offset 3930)
    FOR k := 0 TO 14 DO
        lut_tmp[k] := "NeuroPLC_Weights".w1[3930 + k];
    END_FOR;
    v3[9, 10] := "BsplineEval"(x := v0[10], lut_grid := "NeuroPLC_Weights".w0, lut_table := lut_tmp);
    // φ[11→9]: evaluate LUT (table offset 3945)
    FOR k := 0 TO 14 DO
        lut_tmp[k] := "NeuroPLC_Weights".w1[3945 + k];
    END_FOR;
    v3[9, 11] := "BsplineEval"(x := v0[11], lut_grid := "NeuroPLC_Weights".w0, lut_table := lut_tmp);
    // φ[12→9]: evaluate LUT (table offset 3960)
    FOR k := 0 TO 14 DO
        lut_tmp[k] := "NeuroPLC_Weights".w1[3960 + k];
    END_FOR;
    v3[9, 12] := "BsplineEval"(x := v0[12], lut_grid := "NeuroPLC_Weights".w0, lut_table := lut_tmp);
    // φ[13→9]: evaluate LUT (table offset 3975)
    FOR k := 0 TO 14 DO
        lut_tmp[k] := "NeuroPLC_Weights".w1[3975 + k];
    END_FOR;
    v3[9, 13] := "BsplineEval"(x := v0[13], lut_grid := "NeuroPLC_Weights".w0, lut_table := lut_tmp);
    // φ[14→9]: evaluate LUT (table offset 3990)
    FOR k := 0 TO 14 DO
        lut_tmp[k] := "NeuroPLC_Weights".w1[3990 + k];
    END_FOR;
    v3[9, 14] := "BsplineEval"(x := v0[14], lut_grid := "NeuroPLC_Weights".w0, lut_table := lut_tmp);
    // φ[15→9]: evaluate LUT (table offset 4005)
    FOR k := 0 TO 14 DO
        lut_tmp[k] := "NeuroPLC_Weights".w1[4005 + k];
    END_FOR;
    v3[9, 15] := "BsplineEval"(x := v0[15], lut_grid := "NeuroPLC_Weights".w0, lut_table := lut_tmp);
    // φ[16→9]: evaluate LUT (table offset 4020)
    FOR k := 0 TO 14 DO
        lut_tmp[k] := "NeuroPLC_Weights".w1[4020 + k];
    END_FOR;
    v3[9, 16] := "BsplineEval"(x := v0[16], lut_grid := "NeuroPLC_Weights".w0, lut_table := lut_tmp);
    // φ[17→9]: evaluate LUT (table offset 4035)
    FOR k := 0 TO 14 DO
        lut_tmp[k] := "NeuroPLC_Weights".w1[4035 + k];
    END_FOR;
    v3[9, 17] := "BsplineEval"(x := v0[17], lut_grid := "NeuroPLC_Weights".w0, lut_table := lut_tmp);
    // φ[18→9]: evaluate LUT (table offset 4050)
    FOR k := 0 TO 14 DO
        lut_tmp[k] := "NeuroPLC_Weights".w1[4050 + k];
    END_FOR;
    v3[9, 18] := "BsplineEval"(x := v0[18], lut_grid := "NeuroPLC_Weights".w0, lut_table := lut_tmp);
    // φ[19→9]: evaluate LUT (table offset 4065)
    FOR k := 0 TO 14 DO
        lut_tmp[k] := "NeuroPLC_Weights".w1[4065 + k];
    END_FOR;
    v3[9, 19] := "BsplineEval"(x := v0[19], lut_grid := "NeuroPLC_Weights".w0, lut_table := lut_tmp);
    // φ[20→9]: evaluate LUT (table offset 4080)
    FOR k := 0 TO 14 DO
        lut_tmp[k] := "NeuroPLC_Weights".w1[4080 + k];
    END_FOR;
    v3[9, 20] := "BsplineEval"(x := v0[20], lut_grid := "NeuroPLC_Weights".w0, lut_table := lut_tmp);
    // φ[21→9]: evaluate LUT (table offset 4095)
    FOR k := 0 TO 14 DO
        lut_tmp[k] := "NeuroPLC_Weights".w1[4095 + k];
    END_FOR;
    v3[9, 21] := "BsplineEval"(x := v0[21], lut_grid := "NeuroPLC_Weights".w0, lut_table := lut_tmp);
    // φ[22→9]: evaluate LUT (table offset 4110)
    FOR k := 0 TO 14 DO
        lut_tmp[k] := "NeuroPLC_Weights".w1[4110 + k];
    END_FOR;
    v3[9, 22] := "BsplineEval"(x := v0[22], lut_grid := "NeuroPLC_Weights".w0, lut_table := lut_tmp);
    // φ[23→9]: evaluate LUT (table offset 4125)
    FOR k := 0 TO 14 DO
        lut_tmp[k] := "NeuroPLC_Weights".w1[4125 + k];
    END_FOR;
    v3[9, 23] := "BsplineEval"(x := v0[23], lut_grid := "NeuroPLC_Weights".w0, lut_table := lut_tmp);
    // φ[24→9]: evaluate LUT (table offset 4140)
    FOR k := 0 TO 14 DO
        lut_tmp[k] := "NeuroPLC_Weights".w1[4140 + k];
    END_FOR;
    v3[9, 24] := "BsplineEval"(x := v0[24], lut_grid := "NeuroPLC_Weights".w0, lut_table := lut_tmp);
    // φ[25→9]: evaluate LUT (table offset 4155)
    FOR k := 0 TO 14 DO
        lut_tmp[k] := "NeuroPLC_Weights".w1[4155 + k];
    END_FOR;
    v3[9, 25] := "BsplineEval"(x := v0[25], lut_grid := "NeuroPLC_Weights".w0, lut_table := lut_tmp);
    // φ[26→9]: evaluate LUT (table offset 4170)
    FOR k := 0 TO 14 DO
        lut_tmp[k] := "NeuroPLC_Weights".w1[4170 + k];
    END_FOR;
    v3[9, 26] := "BsplineEval"(x := v0[26], lut_grid := "NeuroPLC_Weights".w0, lut_table := lut_tmp);
    // φ[27→9]: evaluate LUT (table offset 4185)
    FOR k := 0 TO 14 DO
        lut_tmp[k] := "NeuroPLC_Weights".w1[4185 + k];
    END_FOR;
    v3[9, 27] := "BsplineEval"(x := v0[27], lut_grid := "NeuroPLC_Weights".w0, lut_table := lut_tmp);
    // φ[0→10]: evaluate LUT (table offset 4200)
    FOR k := 0 TO 14 DO
        lut_tmp[k] := "NeuroPLC_Weights".w1[4200 + k];
    END_FOR;
    v3[10, 0] := "BsplineEval"(x := v0[0], lut_grid := "NeuroPLC_Weights".w0, lut_table := lut_tmp);
    // φ[1→10]: evaluate LUT (table offset 4215)
    FOR k := 0 TO 14 DO
        lut_tmp[k] := "NeuroPLC_Weights".w1[4215 + k];
    END_FOR;
    v3[10, 1] := "BsplineEval"(x := v0[1], lut_grid := "NeuroPLC_Weights".w0, lut_table := lut_tmp);
    // φ[2→10]: evaluate LUT (table offset 4230)
    FOR k := 0 TO 14 DO
        lut_tmp[k] := "NeuroPLC_Weights".w1[4230 + k];
    END_FOR;
    v3[10, 2] := "BsplineEval"(x := v0[2], lut_grid := "NeuroPLC_Weights".w0, lut_table := lut_tmp);
    // φ[3→10]: evaluate LUT (table offset 4245)
    FOR k := 0 TO 14 DO
        lut_tmp[k] := "NeuroPLC_Weights".w1[4245 + k];
    END_FOR;
    v3[10, 3] := "BsplineEval"(x := v0[3], lut_grid := "NeuroPLC_Weights".w0, lut_table := lut_tmp);
    // φ[4→10]: evaluate LUT (table offset 4260)
    FOR k := 0 TO 14 DO
        lut_tmp[k] := "NeuroPLC_Weights".w1[4260 + k];
    END_FOR;
    v3[10, 4] := "BsplineEval"(x := v0[4], lut_grid := "NeuroPLC_Weights".w0, lut_table := lut_tmp);
    // φ[5→10]: evaluate LUT (table offset 4275)
    FOR k := 0 TO 14 DO
        lut_tmp[k] := "NeuroPLC_Weights".w1[4275 + k];
    END_FOR;
    v3[10, 5] := "BsplineEval"(x := v0[5], lut_grid := "NeuroPLC_Weights".w0, lut_table := lut_tmp);
    // φ[6→10]: evaluate LUT (table offset 4290)
    FOR k := 0 TO 14 DO
        lut_tmp[k] := "NeuroPLC_Weights".w1[4290 + k];
    END_FOR;
    v3[10, 6] := "BsplineEval"(x := v0[6], lut_grid := "NeuroPLC_Weights".w0, lut_table := lut_tmp);
    // φ[7→10]: evaluate LUT (table offset 4305)
    FOR k := 0 TO 14 DO
        lut_tmp[k] := "NeuroPLC_Weights".w1[4305 + k];
    END_FOR;
    v3[10, 7] := "BsplineEval"(x := v0[7], lut_grid := "NeuroPLC_Weights".w0, lut_table := lut_tmp);
    // φ[8→10]: evaluate LUT (table offset 4320)
    FOR k := 0 TO 14 DO
        lut_tmp[k] := "NeuroPLC_Weights".w1[4320 + k];
    END_FOR;
    v3[10, 8] := "BsplineEval"(x := v0[8], lut_grid := "NeuroPLC_Weights".w0, lut_table := lut_tmp);
    // φ[9→10]: evaluate LUT (table offset 4335)
    FOR k := 0 TO 14 DO
        lut_tmp[k] := "NeuroPLC_Weights".w1[4335 + k];
    END_FOR;
    v3[10, 9] := "BsplineEval"(x := v0[9], lut_grid := "NeuroPLC_Weights".w0, lut_table := lut_tmp);
    // φ[10→10]: evaluate LUT (table offset 4350)
    FOR k := 0 TO 14 DO
        lut_tmp[k] := "NeuroPLC_Weights".w1[4350 + k];
    END_FOR;
    v3[10, 10] := "BsplineEval"(x := v0[10], lut_grid := "NeuroPLC_Weights".w0, lut_table := lut_tmp);
    // φ[11→10]: evaluate LUT (table offset 4365)
    FOR k := 0 TO 14 DO
        lut_tmp[k] := "NeuroPLC_Weights".w1[4365 + k];
    END_FOR;
    v3[10, 11] := "BsplineEval"(x := v0[11], lut_grid := "NeuroPLC_Weights".w0, lut_table := lut_tmp);
    // φ[12→10]: evaluate LUT (table offset 4380)
    FOR k := 0 TO 14 DO
        lut_tmp[k] := "NeuroPLC_Weights".w1[4380 + k];
    END_FOR;
    v3[10, 12] := "BsplineEval"(x := v0[12], lut_grid := "NeuroPLC_Weights".w0, lut_table := lut_tmp);
    // φ[13→10]: evaluate LUT (table offset 4395)
    FOR k := 0 TO 14 DO
        lut_tmp[k] := "NeuroPLC_Weights".w1[4395 + k];
    END_FOR;
    v3[10, 13] := "BsplineEval"(x := v0[13], lut_grid := "NeuroPLC_Weights".w0, lut_table := lut_tmp);
    // φ[14→10]: evaluate LUT (table offset 4410)
    FOR k := 0 TO 14 DO
        lut_tmp[k] := "NeuroPLC_Weights".w1[4410 + k];
    END_FOR;
    v3[10, 14] := "BsplineEval"(x := v0[14], lut_grid := "NeuroPLC_Weights".w0, lut_table := lut_tmp);
    // φ[15→10]: evaluate LUT (table offset 4425)
    FOR k := 0 TO 14 DO
        lut_tmp[k] := "NeuroPLC_Weights".w1[4425 + k];
    END_FOR;
    v3[10, 15] := "BsplineEval"(x := v0[15], lut_grid := "NeuroPLC_Weights".w0, lut_table := lut_tmp);
    // φ[16→10]: evaluate LUT (table offset 4440)
    FOR k := 0 TO 14 DO
        lut_tmp[k] := "NeuroPLC_Weights".w1[4440 + k];
    END_FOR;
    v3[10, 16] := "BsplineEval"(x := v0[16], lut_grid := "NeuroPLC_Weights".w0, lut_table := lut_tmp);
    // φ[17→10]: evaluate LUT (table offset 4455)
    FOR k := 0 TO 14 DO
        lut_tmp[k] := "NeuroPLC_Weights".w1[4455 + k];
    END_FOR;
    v3[10, 17] := "BsplineEval"(x := v0[17], lut_grid := "NeuroPLC_Weights".w0, lut_table := lut_tmp);
    // φ[18→10]: evaluate LUT (table offset 4470)
    FOR k := 0 TO 14 DO
        lut_tmp[k] := "NeuroPLC_Weights".w1[4470 + k];
    END_FOR;
    v3[10, 18] := "BsplineEval"(x := v0[18], lut_grid := "NeuroPLC_Weights".w0, lut_table := lut_tmp);
    // φ[19→10]: evaluate LUT (table offset 4485)
    FOR k := 0 TO 14 DO
        lut_tmp[k] := "NeuroPLC_Weights".w1[4485 + k];
    END_FOR;
    v3[10, 19] := "BsplineEval"(x := v0[19], lut_grid := "NeuroPLC_Weights".w0, lut_table := lut_tmp);
    // φ[20→10]: evaluate LUT (table offset 4500)
    FOR k := 0 TO 14 DO
        lut_tmp[k] := "NeuroPLC_Weights".w1[4500 + k];
    END_FOR;
    v3[10, 20] := "BsplineEval"(x := v0[20], lut_grid := "NeuroPLC_Weights".w0, lut_table := lut_tmp);
    // φ[21→10]: evaluate LUT (table offset 4515)
    FOR k := 0 TO 14 DO
        lut_tmp[k] := "NeuroPLC_Weights".w1[4515 + k];
    END_FOR;
    v3[10, 21] := "BsplineEval"(x := v0[21], lut_grid := "NeuroPLC_Weights".w0, lut_table := lut_tmp);
    // φ[22→10]: evaluate LUT (table offset 4530)
    FOR k := 0 TO 14 DO
        lut_tmp[k] := "NeuroPLC_Weights".w1[4530 + k];
    END_FOR;
    v3[10, 22] := "BsplineEval"(x := v0[22], lut_grid := "NeuroPLC_Weights".w0, lut_table := lut_tmp);
    // φ[23→10]: evaluate LUT (table offset 4545)
    FOR k := 0 TO 14 DO
        lut_tmp[k] := "NeuroPLC_Weights".w1[4545 + k];
    END_FOR;
    v3[10, 23] := "BsplineEval"(x := v0[23], lut_grid := "NeuroPLC_Weights".w0, lut_table := lut_tmp);
    // φ[24→10]: evaluate LUT (table offset 4560)
    FOR k := 0 TO 14 DO
        lut_tmp[k] := "NeuroPLC_Weights".w1[4560 + k];
    END_FOR;
    v3[10, 24] := "BsplineEval"(x := v0[24], lut_grid := "NeuroPLC_Weights".w0, lut_table := lut_tmp);
    // φ[25→10]: evaluate LUT (table offset 4575)
    FOR k := 0 TO 14 DO
        lut_tmp[k] := "NeuroPLC_Weights".w1[4575 + k];
    END_FOR;
    v3[10, 25] := "BsplineEval"(x := v0[25], lut_grid := "NeuroPLC_Weights".w0, lut_table := lut_tmp);
    // φ[26→10]: evaluate LUT (table offset 4590)
    FOR k := 0 TO 14 DO
        lut_tmp[k] := "NeuroPLC_Weights".w1[4590 + k];
    END_FOR;
    v3[10, 26] := "BsplineEval"(x := v0[26], lut_grid := "NeuroPLC_Weights".w0, lut_table := lut_tmp);
    // φ[27→10]: evaluate LUT (table offset 4605)
    FOR k := 0 TO 14 DO
        lut_tmp[k] := "NeuroPLC_Weights".w1[4605 + k];
    END_FOR;
    v3[10, 27] := "BsplineEval"(x := v0[27], lut_grid := "NeuroPLC_Weights".w0, lut_table := lut_tmp);
    // φ[0→11]: evaluate LUT (table offset 4620)
    FOR k := 0 TO 14 DO
        lut_tmp[k] := "NeuroPLC_Weights".w1[4620 + k];
    END_FOR;
    v3[11, 0] := "BsplineEval"(x := v0[0], lut_grid := "NeuroPLC_Weights".w0, lut_table := lut_tmp);
    // φ[1→11]: evaluate LUT (table offset 4635)
    FOR k := 0 TO 14 DO
        lut_tmp[k] := "NeuroPLC_Weights".w1[4635 + k];
    END_FOR;
    v3[11, 1] := "BsplineEval"(x := v0[1], lut_grid := "NeuroPLC_Weights".w0, lut_table := lut_tmp);
    // φ[2→11]: evaluate LUT (table offset 4650)
    FOR k := 0 TO 14 DO
        lut_tmp[k] := "NeuroPLC_Weights".w1[4650 + k];
    END_FOR;
    v3[11, 2] := "BsplineEval"(x := v0[2], lut_grid := "NeuroPLC_Weights".w0, lut_table := lut_tmp);
    // φ[3→11]: evaluate LUT (table offset 4665)
    FOR k := 0 TO 14 DO
        lut_tmp[k] := "NeuroPLC_Weights".w1[4665 + k];
    END_FOR;
    v3[11, 3] := "BsplineEval"(x := v0[3], lut_grid := "NeuroPLC_Weights".w0, lut_table := lut_tmp);
    // φ[4→11]: evaluate LUT (table offset 4680)
    FOR k := 0 TO 14 DO
        lut_tmp[k] := "NeuroPLC_Weights".w1[4680 + k];
    END_FOR;
    v3[11, 4] := "BsplineEval"(x := v0[4], lut_grid := "NeuroPLC_Weights".w0, lut_table := lut_tmp);
    // φ[5→11]: evaluate LUT (table offset 4695)
    FOR k := 0 TO 14 DO
        lut_tmp[k] := "NeuroPLC_Weights".w1[4695 + k];
    END_FOR;
    v3[11, 5] := "BsplineEval"(x := v0[5], lut_grid := "NeuroPLC_Weights".w0, lut_table := lut_tmp);
    // φ[6→11]: evaluate LUT (table offset 4710)
    FOR k := 0 TO 14 DO
        lut_tmp[k] := "NeuroPLC_Weights".w1[4710 + k];
    END_FOR;
    v3[11, 6] := "BsplineEval"(x := v0[6], lut_grid := "NeuroPLC_Weights".w0, lut_table := lut_tmp);
    // φ[7→11]: evaluate LUT (table offset 4725)
    FOR k := 0 TO 14 DO
        lut_tmp[k] := "NeuroPLC_Weights".w1[4725 + k];
    END_FOR;
    v3[11, 7] := "BsplineEval"(x := v0[7], lut_grid := "NeuroPLC_Weights".w0, lut_table := lut_tmp);
    // φ[8→11]: evaluate LUT (table offset 4740)
    FOR k := 0 TO 14 DO
        lut_tmp[k] := "NeuroPLC_Weights".w1[4740 + k];
    END_FOR;
    v3[11, 8] := "BsplineEval"(x := v0[8], lut_grid := "NeuroPLC_Weights".w0, lut_table := lut_tmp);
    // φ[9→11]: evaluate LUT (table offset 4755)
    FOR k := 0 TO 14 DO
        lut_tmp[k] := "NeuroPLC_Weights".w1[4755 + k];
    END_FOR;
    v3[11, 9] := "BsplineEval"(x := v0[9], lut_grid := "NeuroPLC_Weights".w0, lut_table := lut_tmp);
    // φ[10→11]: evaluate LUT (table offset 4770)
    FOR k := 0 TO 14 DO
        lut_tmp[k] := "NeuroPLC_Weights".w1[4770 + k];
    END_FOR;
    v3[11, 10] := "BsplineEval"(x := v0[10], lut_grid := "NeuroPLC_Weights".w0, lut_table := lut_tmp);
    // φ[11→11]: evaluate LUT (table offset 4785)
    FOR k := 0 TO 14 DO
        lut_tmp[k] := "NeuroPLC_Weights".w1[4785 + k];
    END_FOR;
    v3[11, 11] := "BsplineEval"(x := v0[11], lut_grid := "NeuroPLC_Weights".w0, lut_table := lut_tmp);
    // φ[12→11]: evaluate LUT (table offset 4800)
    FOR k := 0 TO 14 DO
        lut_tmp[k] := "NeuroPLC_Weights".w1[4800 + k];
    END_FOR;
    v3[11, 12] := "BsplineEval"(x := v0[12], lut_grid := "NeuroPLC_Weights".w0, lut_table := lut_tmp);
    // φ[13→11]: evaluate LUT (table offset 4815)
    FOR k := 0 TO 14 DO
        lut_tmp[k] := "NeuroPLC_Weights".w1[4815 + k];
    END_FOR;
    v3[11, 13] := "BsplineEval"(x := v0[13], lut_grid := "NeuroPLC_Weights".w0, lut_table := lut_tmp);
    // φ[14→11]: evaluate LUT (table offset 4830)
    FOR k := 0 TO 14 DO
        lut_tmp[k] := "NeuroPLC_Weights".w1[4830 + k];
    END_FOR;
    v3[11, 14] := "BsplineEval"(x := v0[14], lut_grid := "NeuroPLC_Weights".w0, lut_table := lut_tmp);
    // φ[15→11]: evaluate LUT (table offset 4845)
    FOR k := 0 TO 14 DO
        lut_tmp[k] := "NeuroPLC_Weights".w1[4845 + k];
    END_FOR;
    v3[11, 15] := "BsplineEval"(x := v0[15], lut_grid := "NeuroPLC_Weights".w0, lut_table := lut_tmp);
    // φ[16→11]: evaluate LUT (table offset 4860)
    FOR k := 0 TO 14 DO
        lut_tmp[k] := "NeuroPLC_Weights".w1[4860 + k];
    END_FOR;
    v3[11, 16] := "BsplineEval"(x := v0[16], lut_grid := "NeuroPLC_Weights".w0, lut_table := lut_tmp);
    // φ[17→11]: evaluate LUT (table offset 4875)
    FOR k := 0 TO 14 DO
        lut_tmp[k] := "NeuroPLC_Weights".w1[4875 + k];
    END_FOR;
    v3[11, 17] := "BsplineEval"(x := v0[17], lut_grid := "NeuroPLC_Weights".w0, lut_table := lut_tmp);
    // φ[18→11]: evaluate LUT (table offset 4890)
    FOR k := 0 TO 14 DO
        lut_tmp[k] := "NeuroPLC_Weights".w1[4890 + k];
    END_FOR;
    v3[11, 18] := "BsplineEval"(x := v0[18], lut_grid := "NeuroPLC_Weights".w0, lut_table := lut_tmp);
    // φ[19→11]: evaluate LUT (table offset 4905)
    FOR k := 0 TO 14 DO
        lut_tmp[k] := "NeuroPLC_Weights".w1[4905 + k];
    END_FOR;
    v3[11, 19] := "BsplineEval"(x := v0[19], lut_grid := "NeuroPLC_Weights".w0, lut_table := lut_tmp);
    // φ[20→11]: evaluate LUT (table offset 4920)
    FOR k := 0 TO 14 DO
        lut_tmp[k] := "NeuroPLC_Weights".w1[4920 + k];
    END_FOR;
    v3[11, 20] := "BsplineEval"(x := v0[20], lut_grid := "NeuroPLC_Weights".w0, lut_table := lut_tmp);
    // φ[21→11]: evaluate LUT (table offset 4935)
    FOR k := 0 TO 14 DO
        lut_tmp[k] := "NeuroPLC_Weights".w1[4935 + k];
    END_FOR;
    v3[11, 21] := "BsplineEval"(x := v0[21], lut_grid := "NeuroPLC_Weights".w0, lut_table := lut_tmp);
    // φ[22→11]: evaluate LUT (table offset 4950)
    FOR k := 0 TO 14 DO
        lut_tmp[k] := "NeuroPLC_Weights".w1[4950 + k];
    END_FOR;
    v3[11, 22] := "BsplineEval"(x := v0[22], lut_grid := "NeuroPLC_Weights".w0, lut_table := lut_tmp);
    // φ[23→11]: evaluate LUT (table offset 4965)
    FOR k := 0 TO 14 DO
        lut_tmp[k] := "NeuroPLC_Weights".w1[4965 + k];
    END_FOR;
    v3[11, 23] := "BsplineEval"(x := v0[23], lut_grid := "NeuroPLC_Weights".w0, lut_table := lut_tmp);
    // φ[24→11]: evaluate LUT (table offset 4980)
    FOR k := 0 TO 14 DO
        lut_tmp[k] := "NeuroPLC_Weights".w1[4980 + k];
    END_FOR;
    v3[11, 24] := "BsplineEval"(x := v0[24], lut_grid := "NeuroPLC_Weights".w0, lut_table := lut_tmp);
    // φ[25→11]: evaluate LUT (table offset 4995)
    FOR k := 0 TO 14 DO
        lut_tmp[k] := "NeuroPLC_Weights".w1[4995 + k];
    END_FOR;
    v3[11, 25] := "BsplineEval"(x := v0[25], lut_grid := "NeuroPLC_Weights".w0, lut_table := lut_tmp);
    // φ[26→11]: evaluate LUT (table offset 5010)
    FOR k := 0 TO 14 DO
        lut_tmp[k] := "NeuroPLC_Weights".w1[5010 + k];
    END_FOR;
    v3[11, 26] := "BsplineEval"(x := v0[26], lut_grid := "NeuroPLC_Weights".w0, lut_table := lut_tmp);
    // φ[27→11]: evaluate LUT (table offset 5025)
    FOR k := 0 TO 14 DO
        lut_tmp[k] := "NeuroPLC_Weights".w1[5025 + k];
    END_FOR;
    v3[11, 27] := "BsplineEval"(x := v0[27], lut_grid := "NeuroPLC_Weights".w0, lut_table := lut_tmp);
    // φ[0→12]: evaluate LUT (table offset 5040)
    FOR k := 0 TO 14 DO
        lut_tmp[k] := "NeuroPLC_Weights".w1[5040 + k];
    END_FOR;
    v3[12, 0] := "BsplineEval"(x := v0[0], lut_grid := "NeuroPLC_Weights".w0, lut_table := lut_tmp);
    // φ[1→12]: evaluate LUT (table offset 5055)
    FOR k := 0 TO 14 DO
        lut_tmp[k] := "NeuroPLC_Weights".w1[5055 + k];
    END_FOR;
    v3[12, 1] := "BsplineEval"(x := v0[1], lut_grid := "NeuroPLC_Weights".w0, lut_table := lut_tmp);
    // φ[2→12]: evaluate LUT (table offset 5070)
    FOR k := 0 TO 14 DO
        lut_tmp[k] := "NeuroPLC_Weights".w1[5070 + k];
    END_FOR;
    v3[12, 2] := "BsplineEval"(x := v0[2], lut_grid := "NeuroPLC_Weights".w0, lut_table := lut_tmp);
    // φ[3→12]: evaluate LUT (table offset 5085)
    FOR k := 0 TO 14 DO
        lut_tmp[k] := "NeuroPLC_Weights".w1[5085 + k];
    END_FOR;
    v3[12, 3] := "BsplineEval"(x := v0[3], lut_grid := "NeuroPLC_Weights".w0, lut_table := lut_tmp);
    // φ[4→12]: evaluate LUT (table offset 5100)
    FOR k := 0 TO 14 DO
        lut_tmp[k] := "NeuroPLC_Weights".w1[5100 + k];
    END_FOR;
    v3[12, 4] := "BsplineEval"(x := v0[4], lut_grid := "NeuroPLC_Weights".w0, lut_table := lut_tmp);
    // φ[5→12]: evaluate LUT (table offset 5115)
    FOR k := 0 TO 14 DO
        lut_tmp[k] := "NeuroPLC_Weights".w1[5115 + k];
    END_FOR;
    v3[12, 5] := "BsplineEval"(x := v0[5], lut_grid := "NeuroPLC_Weights".w0, lut_table := lut_tmp);
    // φ[6→12]: evaluate LUT (table offset 5130)
    FOR k := 0 TO 14 DO
        lut_tmp[k] := "NeuroPLC_Weights".w1[5130 + k];
    END_FOR;
    v3[12, 6] := "BsplineEval"(x := v0[6], lut_grid := "NeuroPLC_Weights".w0, lut_table := lut_tmp);
    // φ[7→12]: evaluate LUT (table offset 5145)
    FOR k := 0 TO 14 DO
        lut_tmp[k] := "NeuroPLC_Weights".w1[5145 + k];
    END_FOR;
    v3[12, 7] := "BsplineEval"(x := v0[7], lut_grid := "NeuroPLC_Weights".w0, lut_table := lut_tmp);
    // φ[8→12]: evaluate LUT (table offset 5160)
    FOR k := 0 TO 14 DO
        lut_tmp[k] := "NeuroPLC_Weights".w1[5160 + k];
    END_FOR;
    v3[12, 8] := "BsplineEval"(x := v0[8], lut_grid := "NeuroPLC_Weights".w0, lut_table := lut_tmp);
    // φ[9→12]: evaluate LUT (table offset 5175)
    FOR k := 0 TO 14 DO
        lut_tmp[k] := "NeuroPLC_Weights".w1[5175 + k];
    END_FOR;
    v3[12, 9] := "BsplineEval"(x := v0[9], lut_grid := "NeuroPLC_Weights".w0, lut_table := lut_tmp);
    // φ[10→12]: evaluate LUT (table offset 5190)
    FOR k := 0 TO 14 DO
        lut_tmp[k] := "NeuroPLC_Weights".w1[5190 + k];
    END_FOR;
    v3[12, 10] := "BsplineEval"(x := v0[10], lut_grid := "NeuroPLC_Weights".w0, lut_table := lut_tmp);
    // φ[11→12]: evaluate LUT (table offset 5205)
    FOR k := 0 TO 14 DO
        lut_tmp[k] := "NeuroPLC_Weights".w1[5205 + k];
    END_FOR;
    v3[12, 11] := "BsplineEval"(x := v0[11], lut_grid := "NeuroPLC_Weights".w0, lut_table := lut_tmp);
    // φ[12→12]: evaluate LUT (table offset 5220)
    FOR k := 0 TO 14 DO
        lut_tmp[k] := "NeuroPLC_Weights".w1[5220 + k];
    END_FOR;
    v3[12, 12] := "BsplineEval"(x := v0[12], lut_grid := "NeuroPLC_Weights".w0, lut_table := lut_tmp);
    // φ[13→12]: evaluate LUT (table offset 5235)
    FOR k := 0 TO 14 DO
        lut_tmp[k] := "NeuroPLC_Weights".w1[5235 + k];
    END_FOR;
    v3[12, 13] := "BsplineEval"(x := v0[13], lut_grid := "NeuroPLC_Weights".w0, lut_table := lut_tmp);
    // φ[14→12]: evaluate LUT (table offset 5250)
    FOR k := 0 TO 14 DO
        lut_tmp[k] := "NeuroPLC_Weights".w1[5250 + k];
    END_FOR;
    v3[12, 14] := "BsplineEval"(x := v0[14], lut_grid := "NeuroPLC_Weights".w0, lut_table := lut_tmp);
    // φ[15→12]: evaluate LUT (table offset 5265)
    FOR k := 0 TO 14 DO
        lut_tmp[k] := "NeuroPLC_Weights".w1[5265 + k];
    END_FOR;
    v3[12, 15] := "BsplineEval"(x := v0[15], lut_grid := "NeuroPLC_Weights".w0, lut_table := lut_tmp);
    // φ[16→12]: evaluate LUT (table offset 5280)
    FOR k := 0 TO 14 DO
        lut_tmp[k] := "NeuroPLC_Weights".w1[5280 + k];
    END_FOR;
    v3[12, 16] := "BsplineEval"(x := v0[16], lut_grid := "NeuroPLC_Weights".w0, lut_table := lut_tmp);
    // φ[17→12]: evaluate LUT (table offset 5295)
    FOR k := 0 TO 14 DO
        lut_tmp[k] := "NeuroPLC_Weights".w1[5295 + k];
    END_FOR;
    v3[12, 17] := "BsplineEval"(x := v0[17], lut_grid := "NeuroPLC_Weights".w0, lut_table := lut_tmp);
    // φ[18→12]: evaluate LUT (table offset 5310)
    FOR k := 0 TO 14 DO
        lut_tmp[k] := "NeuroPLC_Weights".w1[5310 + k];
    END_FOR;
    v3[12, 18] := "BsplineEval"(x := v0[18], lut_grid := "NeuroPLC_Weights".w0, lut_table := lut_tmp);
    // φ[19→12]: evaluate LUT (table offset 5325)
    FOR k := 0 TO 14 DO
        lut_tmp[k] := "NeuroPLC_Weights".w1[5325 + k];
    END_FOR;
    v3[12, 19] := "BsplineEval"(x := v0[19], lut_grid := "NeuroPLC_Weights".w0, lut_table := lut_tmp);
    // φ[20→12]: evaluate LUT (table offset 5340)
    FOR k := 0 TO 14 DO
        lut_tmp[k] := "NeuroPLC_Weights".w1[5340 + k];
    END_FOR;
    v3[12, 20] := "BsplineEval"(x := v0[20], lut_grid := "NeuroPLC_Weights".w0, lut_table := lut_tmp);
    // φ[21→12]: evaluate LUT (table offset 5355)
    FOR k := 0 TO 14 DO
        lut_tmp[k] := "NeuroPLC_Weights".w1[5355 + k];
    END_FOR;
    v3[12, 21] := "BsplineEval"(x := v0[21], lut_grid := "NeuroPLC_Weights".w0, lut_table := lut_tmp);
    // φ[22→12]: evaluate LUT (table offset 5370)
    FOR k := 0 TO 14 DO
        lut_tmp[k] := "NeuroPLC_Weights".w1[5370 + k];
    END_FOR;
    v3[12, 22] := "BsplineEval"(x := v0[22], lut_grid := "NeuroPLC_Weights".w0, lut_table := lut_tmp);
    // φ[23→12]: evaluate LUT (table offset 5385)
    FOR k := 0 TO 14 DO
        lut_tmp[k] := "NeuroPLC_Weights".w1[5385 + k];
    END_FOR;
    v3[12, 23] := "BsplineEval"(x := v0[23], lut_grid := "NeuroPLC_Weights".w0, lut_table := lut_tmp);
    // φ[24→12]: evaluate LUT (table offset 5400)
    FOR k := 0 TO 14 DO
        lut_tmp[k] := "NeuroPLC_Weights".w1[5400 + k];
    END_FOR;
    v3[12, 24] := "BsplineEval"(x := v0[24], lut_grid := "NeuroPLC_Weights".w0, lut_table := lut_tmp);
    // φ[25→12]: evaluate LUT (table offset 5415)
    FOR k := 0 TO 14 DO
        lut_tmp[k] := "NeuroPLC_Weights".w1[5415 + k];
    END_FOR;
    v3[12, 25] := "BsplineEval"(x := v0[25], lut_grid := "NeuroPLC_Weights".w0, lut_table := lut_tmp);
    // φ[26→12]: evaluate LUT (table offset 5430)
    FOR k := 0 TO 14 DO
        lut_tmp[k] := "NeuroPLC_Weights".w1[5430 + k];
    END_FOR;
    v3[12, 26] := "BsplineEval"(x := v0[26], lut_grid := "NeuroPLC_Weights".w0, lut_table := lut_tmp);
    // φ[27→12]: evaluate LUT (table offset 5445)
    FOR k := 0 TO 14 DO
        lut_tmp[k] := "NeuroPLC_Weights".w1[5445 + k];
    END_FOR;
    v3[12, 27] := "BsplineEval"(x := v0[27], lut_grid := "NeuroPLC_Weights".w0, lut_table := lut_tmp);
    // φ[0→13]: evaluate LUT (table offset 5460)
    FOR k := 0 TO 14 DO
        lut_tmp[k] := "NeuroPLC_Weights".w1[5460 + k];
    END_FOR;
    v3[13, 0] := "BsplineEval"(x := v0[0], lut_grid := "NeuroPLC_Weights".w0, lut_table := lut_tmp);
    // φ[1→13]: evaluate LUT (table offset 5475)
    FOR k := 0 TO 14 DO
        lut_tmp[k] := "NeuroPLC_Weights".w1[5475 + k];
    END_FOR;
    v3[13, 1] := "BsplineEval"(x := v0[1], lut_grid := "NeuroPLC_Weights".w0, lut_table := lut_tmp);
    // φ[2→13]: evaluate LUT (table offset 5490)
    FOR k := 0 TO 14 DO
        lut_tmp[k] := "NeuroPLC_Weights".w1[5490 + k];
    END_FOR;
    v3[13, 2] := "BsplineEval"(x := v0[2], lut_grid := "NeuroPLC_Weights".w0, lut_table := lut_tmp);
    // φ[3→13]: evaluate LUT (table offset 5505)
    FOR k := 0 TO 14 DO
        lut_tmp[k] := "NeuroPLC_Weights".w1[5505 + k];
    END_FOR;
    v3[13, 3] := "BsplineEval"(x := v0[3], lut_grid := "NeuroPLC_Weights".w0, lut_table := lut_tmp);
    // φ[4→13]: evaluate LUT (table offset 5520)
    FOR k := 0 TO 14 DO
        lut_tmp[k] := "NeuroPLC_Weights".w1[5520 + k];
    END_FOR;
    v3[13, 4] := "BsplineEval"(x := v0[4], lut_grid := "NeuroPLC_Weights".w0, lut_table := lut_tmp);
    // φ[5→13]: evaluate LUT (table offset 5535)
    FOR k := 0 TO 14 DO
        lut_tmp[k] := "NeuroPLC_Weights".w1[5535 + k];
    END_FOR;
    v3[13, 5] := "BsplineEval"(x := v0[5], lut_grid := "NeuroPLC_Weights".w0, lut_table := lut_tmp);
    // φ[6→13]: evaluate LUT (table offset 5550)
    FOR k := 0 TO 14 DO
        lut_tmp[k] := "NeuroPLC_Weights".w1[5550 + k];
    END_FOR;
    v3[13, 6] := "BsplineEval"(x := v0[6], lut_grid := "NeuroPLC_Weights".w0, lut_table := lut_tmp);
    // φ[7→13]: evaluate LUT (table offset 5565)
    FOR k := 0 TO 14 DO
        lut_tmp[k] := "NeuroPLC_Weights".w1[5565 + k];
    END_FOR;
    v3[13, 7] := "BsplineEval"(x := v0[7], lut_grid := "NeuroPLC_Weights".w0, lut_table := lut_tmp);
    // φ[8→13]: evaluate LUT (table offset 5580)
    FOR k := 0 TO 14 DO
        lut_tmp[k] := "NeuroPLC_Weights".w1[5580 + k];
    END_FOR;
    v3[13, 8] := "BsplineEval"(x := v0[8], lut_grid := "NeuroPLC_Weights".w0, lut_table := lut_tmp);
    // φ[9→13]: evaluate LUT (table offset 5595)
    FOR k := 0 TO 14 DO
        lut_tmp[k] := "NeuroPLC_Weights".w1[5595 + k];
    END_FOR;
    v3[13, 9] := "BsplineEval"(x := v0[9], lut_grid := "NeuroPLC_Weights".w0, lut_table := lut_tmp);
    // φ[10→13]: evaluate LUT (table offset 5610)
    FOR k := 0 TO 14 DO
        lut_tmp[k] := "NeuroPLC_Weights".w1[5610 + k];
    END_FOR;
    v3[13, 10] := "BsplineEval"(x := v0[10], lut_grid := "NeuroPLC_Weights".w0, lut_table := lut_tmp);
    // φ[11→13]: evaluate LUT (table offset 5625)
    FOR k := 0 TO 14 DO
        lut_tmp[k] := "NeuroPLC_Weights".w1[5625 + k];
    END_FOR;
    v3[13, 11] := "BsplineEval"(x := v0[11], lut_grid := "NeuroPLC_Weights".w0, lut_table := lut_tmp);
    // φ[12→13]: evaluate LUT (table offset 5640)
    FOR k := 0 TO 14 DO
        lut_tmp[k] := "NeuroPLC_Weights".w1[5640 + k];
    END_FOR;
    v3[13, 12] := "BsplineEval"(x := v0[12], lut_grid := "NeuroPLC_Weights".w0, lut_table := lut_tmp);
    // φ[13→13]: evaluate LUT (table offset 5655)
    FOR k := 0 TO 14 DO
        lut_tmp[k] := "NeuroPLC_Weights".w1[5655 + k];
    END_FOR;
    v3[13, 13] := "BsplineEval"(x := v0[13], lut_grid := "NeuroPLC_Weights".w0, lut_table := lut_tmp);
    // φ[14→13]: evaluate LUT (table offset 5670)
    FOR k := 0 TO 14 DO
        lut_tmp[k] := "NeuroPLC_Weights".w1[5670 + k];
    END_FOR;
    v3[13, 14] := "BsplineEval"(x := v0[14], lut_grid := "NeuroPLC_Weights".w0, lut_table := lut_tmp);
    // φ[15→13]: evaluate LUT (table offset 5685)
    FOR k := 0 TO 14 DO
        lut_tmp[k] := "NeuroPLC_Weights".w1[5685 + k];
    END_FOR;
    v3[13, 15] := "BsplineEval"(x := v0[15], lut_grid := "NeuroPLC_Weights".w0, lut_table := lut_tmp);
    // φ[16→13]: evaluate LUT (table offset 5700)
    FOR k := 0 TO 14 DO
        lut_tmp[k] := "NeuroPLC_Weights".w1[5700 + k];
    END_FOR;
    v3[13, 16] := "BsplineEval"(x := v0[16], lut_grid := "NeuroPLC_Weights".w0, lut_table := lut_tmp);
    // φ[17→13]: evaluate LUT (table offset 5715)
    FOR k := 0 TO 14 DO
        lut_tmp[k] := "NeuroPLC_Weights".w1[5715 + k];
    END_FOR;
    v3[13, 17] := "BsplineEval"(x := v0[17], lut_grid := "NeuroPLC_Weights".w0, lut_table := lut_tmp);
    // φ[18→13]: evaluate LUT (table offset 5730)
    FOR k := 0 TO 14 DO
        lut_tmp[k] := "NeuroPLC_Weights".w1[5730 + k];
    END_FOR;
    v3[13, 18] := "BsplineEval"(x := v0[18], lut_grid := "NeuroPLC_Weights".w0, lut_table := lut_tmp);
    // φ[19→13]: evaluate LUT (table offset 5745)
    FOR k := 0 TO 14 DO
        lut_tmp[k] := "NeuroPLC_Weights".w1[5745 + k];
    END_FOR;
    v3[13, 19] := "BsplineEval"(x := v0[19], lut_grid := "NeuroPLC_Weights".w0, lut_table := lut_tmp);
    // φ[20→13]: evaluate LUT (table offset 5760)
    FOR k := 0 TO 14 DO
        lut_tmp[k] := "NeuroPLC_Weights".w1[5760 + k];
    END_FOR;
    v3[13, 20] := "BsplineEval"(x := v0[20], lut_grid := "NeuroPLC_Weights".w0, lut_table := lut_tmp);
    // φ[21→13]: evaluate LUT (table offset 5775)
    FOR k := 0 TO 14 DO
        lut_tmp[k] := "NeuroPLC_Weights".w1[5775 + k];
    END_FOR;
    v3[13, 21] := "BsplineEval"(x := v0[21], lut_grid := "NeuroPLC_Weights".w0, lut_table := lut_tmp);
    // φ[22→13]: evaluate LUT (table offset 5790)
    FOR k := 0 TO 14 DO
        lut_tmp[k] := "NeuroPLC_Weights".w1[5790 + k];
    END_FOR;
    v3[13, 22] := "BsplineEval"(x := v0[22], lut_grid := "NeuroPLC_Weights".w0, lut_table := lut_tmp);
    // φ[23→13]: evaluate LUT (table offset 5805)
    FOR k := 0 TO 14 DO
        lut_tmp[k] := "NeuroPLC_Weights".w1[5805 + k];
    END_FOR;
    v3[13, 23] := "BsplineEval"(x := v0[23], lut_grid := "NeuroPLC_Weights".w0, lut_table := lut_tmp);
    // φ[24→13]: evaluate LUT (table offset 5820)
    FOR k := 0 TO 14 DO
        lut_tmp[k] := "NeuroPLC_Weights".w1[5820 + k];
    END_FOR;
    v3[13, 24] := "BsplineEval"(x := v0[24], lut_grid := "NeuroPLC_Weights".w0, lut_table := lut_tmp);
    // φ[25→13]: evaluate LUT (table offset 5835)
    FOR k := 0 TO 14 DO
        lut_tmp[k] := "NeuroPLC_Weights".w1[5835 + k];
    END_FOR;
    v3[13, 25] := "BsplineEval"(x := v0[25], lut_grid := "NeuroPLC_Weights".w0, lut_table := lut_tmp);
    // φ[26→13]: evaluate LUT (table offset 5850)
    FOR k := 0 TO 14 DO
        lut_tmp[k] := "NeuroPLC_Weights".w1[5850 + k];
    END_FOR;
    v3[13, 26] := "BsplineEval"(x := v0[26], lut_grid := "NeuroPLC_Weights".w0, lut_table := lut_tmp);
    // φ[27→13]: evaluate LUT (table offset 5865)
    FOR k := 0 TO 14 DO
        lut_tmp[k] := "NeuroPLC_Weights".w1[5865 + k];
    END_FOR;
    v3[13, 27] := "BsplineEval"(x := v0[27], lut_grid := "NeuroPLC_Weights".w0, lut_table := lut_tmp);
    // φ[0→14]: evaluate LUT (table offset 5880)
    FOR k := 0 TO 14 DO
        lut_tmp[k] := "NeuroPLC_Weights".w1[5880 + k];
    END_FOR;
    v3[14, 0] := "BsplineEval"(x := v0[0], lut_grid := "NeuroPLC_Weights".w0, lut_table := lut_tmp);
    // φ[1→14]: evaluate LUT (table offset 5895)
    FOR k := 0 TO 14 DO
        lut_tmp[k] := "NeuroPLC_Weights".w1[5895 + k];
    END_FOR;
    v3[14, 1] := "BsplineEval"(x := v0[1], lut_grid := "NeuroPLC_Weights".w0, lut_table := lut_tmp);
    // φ[2→14]: evaluate LUT (table offset 5910)
    FOR k := 0 TO 14 DO
        lut_tmp[k] := "NeuroPLC_Weights".w1[5910 + k];
    END_FOR;
    v3[14, 2] := "BsplineEval"(x := v0[2], lut_grid := "NeuroPLC_Weights".w0, lut_table := lut_tmp);
    // φ[3→14]: evaluate LUT (table offset 5925)
    FOR k := 0 TO 14 DO
        lut_tmp[k] := "NeuroPLC_Weights".w1[5925 + k];
    END_FOR;
    v3[14, 3] := "BsplineEval"(x := v0[3], lut_grid := "NeuroPLC_Weights".w0, lut_table := lut_tmp);
    // φ[4→14]: evaluate LUT (table offset 5940)
    FOR k := 0 TO 14 DO
        lut_tmp[k] := "NeuroPLC_Weights".w1[5940 + k];
    END_FOR;
    v3[14, 4] := "BsplineEval"(x := v0[4], lut_grid := "NeuroPLC_Weights".w0, lut_table := lut_tmp);
    // φ[5→14]: evaluate LUT (table offset 5955)
    FOR k := 0 TO 14 DO
        lut_tmp[k] := "NeuroPLC_Weights".w1[5955 + k];
    END_FOR;
    v3[14, 5] := "BsplineEval"(x := v0[5], lut_grid := "NeuroPLC_Weights".w0, lut_table := lut_tmp);
    // φ[6→14]: evaluate LUT (table offset 5970)
    FOR k := 0 TO 14 DO
        lut_tmp[k] := "NeuroPLC_Weights".w1[5970 + k];
    END_FOR;
    v3[14, 6] := "BsplineEval"(x := v0[6], lut_grid := "NeuroPLC_Weights".w0, lut_table := lut_tmp);
    // φ[7→14]: evaluate LUT (table offset 5985)
    FOR k := 0 TO 14 DO
        lut_tmp[k] := "NeuroPLC_Weights".w1[5985 + k];
    END_FOR;
    v3[14, 7] := "BsplineEval"(x := v0[7], lut_grid := "NeuroPLC_Weights".w0, lut_table := lut_tmp);
    // φ[8→14]: evaluate LUT (table offset 6000)
    FOR k := 0 TO 14 DO
        lut_tmp[k] := "NeuroPLC_Weights".w1[6000 + k];
    END_FOR;
    v3[14, 8] := "BsplineEval"(x := v0[8], lut_grid := "NeuroPLC_Weights".w0, lut_table := lut_tmp);
    // φ[9→14]: evaluate LUT (table offset 6015)
    FOR k := 0 TO 14 DO
        lut_tmp[k] := "NeuroPLC_Weights".w1[6015 + k];
    END_FOR;
    v3[14, 9] := "BsplineEval"(x := v0[9], lut_grid := "NeuroPLC_Weights".w0, lut_table := lut_tmp);
    // φ[10→14]: evaluate LUT (table offset 6030)
    FOR k := 0 TO 14 DO
        lut_tmp[k] := "NeuroPLC_Weights".w1[6030 + k];
    END_FOR;
    v3[14, 10] := "BsplineEval"(x := v0[10], lut_grid := "NeuroPLC_Weights".w0, lut_table := lut_tmp);
    // φ[11→14]: evaluate LUT (table offset 6045)
    FOR k := 0 TO 14 DO
        lut_tmp[k] := "NeuroPLC_Weights".w1[6045 + k];
    END_FOR;
